# B&R Automation Studio project NAELD004C00R10L518F00 (part 22)

#### Visu_Layer.typ
```iecst
(*Common Layers*)

TYPE
	tyLyrC0001MotionStd : 	STRUCT
		tyBitmapOrigin : tyUIBitmap;
		tyBitmapPwr : tyUIBitmap;
		tyBitmapRst : tyUIBitmap;
		tyBitmapStop : tyUIBitmap;
		tyBitmapMc : tyUIBitmap;
		tyBtnPosLmtSen : tyUIBtn;
		tyBtnNegLmtSen : tyUIBtn;
		tyBtnJogPos : tyUIBtn;
		tyBtnJogNeg : tyUIBtn;
		tyBtnMovAbs : tyUIBtn;
		tyBtnMovRel : tyUIBtn;
		tyBtnOrigin : tyUIBtn;
		tyBtnPwr : tyUIBtn;
		tyBtnRst : tyUIBtn;
		tyBtnStop : tyUIBtn;
		tyNumCurrPos : tyUINum;
		tyNumErrCode : tyUINum;
		tyNumNomSpd : tyUINum;
		tyNumSlwSpd : tyUINum;
		tyNumStepSize : tyUINum;
		tyNumTargetPos : tyUINum;
		tyStringStat : tyUILString;
	END_STRUCT;
	tyLyrC0001MotionStdAW : 	STRUCT
		tyBitmapOrigin : tyUIBitmap;
		tyBitmapPwr : tyUIBitmap;
		tyBitmapRst : tyUIBitmap;
		tyBitmapStop : tyUIBitmap;
		tyBitmapMc : tyUIBitmap;
		tyBtnOpenLmtSen : tyUIBtn;
		tyBtnCloseLmtSen : tyUIBtn;
		tyBtnJogOpen : tyUIBtn;
		tyBtnJogClose : tyUIBtn;
		tyBtnMovAbs : tyUIBtn;
		tyBtnMovRel : tyUIBtn;
		tyBtnOrigin : tyUIBtn;
		tyBtnPwr : tyUIBtn;
		tyBtnRst : tyUIBtn;
		tyBtnStop : tyUIBtn;
		tyNumCurrPos : tyUINum;
		tyNumErrCode : tyUINum;
		tyNumNomSpd : tyUINum;
		tyNumSlwSpd : tyUINum;
		tyNumStepSize : tyUINum;
		tyNumTargetPos : tyUINum;
		tyStringStat : tyUILString;
	END_STRUCT;
	tyLyrC0001MotionStdLifter : 	STRUCT
		tyBitmapOrigin : tyUIBitmap;
		tyBitmapPwr : tyUIBitmap;
		tyBitmapRst : tyUIBitmap;
		tyBitmapStop : tyUIBitmap;
		tyBitmapMc : tyUIBitmap;
		tyBtnUpLmtSen : tyUIBtn;
		tyBtnDownLmtSen : tyUIBtn;
		tyBtnJogUp : tyUIBtn;
		tyBtnJogDown : tyUIBtn;
		tyBtnMovAbs : tyUIBtn;
		tyBtnMovRel : tyUIBtn;
		tyBtnOrigin : tyUIBtn;
		tyBtnPwr : tyUIBtn;
		tyBtnRst : tyUIBtn;
		tyBtnStop : tyUIBtn;
		tyNumCurrPos : tyUINum;
		tyNumErrCode : tyUINum;
		tyNumNomSpd : tyUINum;
		tyNumSlwSpd : tyUINum;
		tyNumStepSize : tyUINum;
		tyNumTargetPos : tyUINum;
		tyStringStat : tyUILString;
	END_STRUCT;
	tyLyrC0001MotionStdTrav : 	STRUCT
		tyBitmapOrigin : tyUIBitmap;
		tyBitmapPwr : tyUIBitmap;
		tyBitmapRst : tyUIBitmap;
		tyBitmapStop : tyUIBitmap;
		tyBitmapMc : tyUIBitmap;
		tyBtnFrontLmtSen : tyUIBtn;
		tyBtnRearLmtSen : tyUIBtn;
		tyBtnJogFront : tyUIBtn;
		tyBtnJogRear : tyUIBtn;
		tyBtnMovAbs : tyUIBtn;
		tyBtnMovRel : tyUIBtn;
		tyBtnOrigin : tyUIBtn;
		tyBtnPwr : tyUIBtn;
		tyBtnRst : tyUIBtn;
		tyBtnStop : tyUIBtn;
		tyNumCurrPos : tyUINum;
		tyNumErrCode : tyUINum;
		tyNumNomSpd : tyUINum;
		tyNumSlwSpd : tyUINum;
		tyNumStepSize : tyUINum;
		tyNumTargetPos : tyUINum;
		tyStringStat : tyUILString;
	END_STRUCT;
	tyLyrC0002FullMask : 	STRUCT
		tyLyr : tyUILyr;
		tyBtnMask : tyUIBtn;
	END_STRUCT;
	tyLyrC0003DualMask : 	STRUCT
		tyBtnLeftMask : tyUIBtn;
		tyBtnRgtMask : tyUIBtn;
		tyLyr : tyUILyr;
	END_STRUCT;
	tyLyrC0004Navi : 	STRUCT
		tyBtnLeft : tyUIBtn;
		tyBtnRgt : tyUIBtn;
		tyBtnBack : tyUIBtn;
		tyBitmapPageDisp : tyUIBitmap;
		tyLyr : tyUILyr;
	END_STRUCT;
	tyLyrC0005Main : 	STRUCT
		tyBtnNotification : tyUIBtn;
		tyBtnHome : tyUIBtn;
		tyBtnBuzzer : tyUIBtn;
		tyBtnStart : tyUIBtn;
		tyBtnStop : tyUIBtn;
		tyBtnStep : tyUIBtn;
		tyBtnReset : tyUIBtn;
		tyBitmapStatBar : tyUIBitmap;
		tyHotspotNaviStart : tyUIHotspot;
		tyBtnAlarm : tyUIBtn;
	END_STRUCT;
	tyLyrC0006Set : 	STRUCT
		tyBtnSave : tyUIBtn;
		tyLyr : tyUILyr;
	END_STRUCT;
	tyLyrC0007Notif : 	STRUCT
		tyTxtUsrLv : tyUITxt;
		tyTxtLFMc : tyUITxt;
		tyHotspotClose : tyUIHotspot;
		tyStringUsrNm : tyUIString;
		tyHotspotShowInfo : tyUIHotspot;
		tyBitmapShowInfo : tyUIBitmap;
		tyLyr : tyUILyr;
	END_STRUCT;
	tyLyrC0008MsgBox : 	STRUCT
		tyBitmapIcon : tyUIBitmap;
		tyBtnNo : tyUIBtn;
		tyBtnYes : tyUIBtn;
		tyLyr : tyUILyr;
		tyTxtWO_sLogMessage : tyUILString;
		tyTxtMsg : tyUITxt;
		tyTxtTitle : tyUITxt;
	END_STRUCT;
	tyLyrC0009Info : 	STRUCT
		tyStringInfo : tyUILString;
		tyHotspotClose : tyUIHotspot;
		tyLyr : tyUILyr;
	END_STRUCT;
	tyLyrC0010RcyMsg : 	STRUCT
		tyTxtMsg : tyUILString;
		tyHotspotClose : tyUIHotspot;
		tyLyr : tyUILyr;
	END_STRUCT;
	tyLyrC0011RcpPopUp : 	STRUCT
		tyStringInfo : tyUILString;
		tyHotspotClose : tyUIHotspot;
		tyLyr : tyUILyr;
	END_STRUCT;
END_TYPE

(**)
(**)
(*Pages*)

TYPE
	tyLyrP0000SSaver : 	STRUCT
		tyTxtMcStat : tyUITxt;
		tyTxtMcNm : tyUILString;
		tyBitmapStat : tyUIBitmap;
	END_STRUCT;
END_TYPE

(**)

TYPE
	tyLyrP0001Startup : 	STRUCT
		tyBarGraphStartup : tyUIBarGraph;
		tyTxtStartupStat : tyUITxt;
	END_STRUCT;
	tyLyrP0001Initial : 	STRUCT
		tyLyr : tyUILyr;
	END_STRUCT;
END_TYPE

(**)

TYPE
	tyLyrP0002Menu : 	STRUCT
		tyBtnAlm : tyUIBtn;
		tyBtnCommCtrl : tyUIBtn;
		tyBtnGenInput : tyUIBtn;
		tyBtnGenOutput : tyUIBtn;
		tyBtnLang : tyUIBtn;
		tyBtnLFCtrl : tyUIBtn;
		tyBtnLFSet : tyUIBtn;
		tyBtnLogin : tyUIBtn;
		tyBtnMcInfo : tyUIBtn;
		tyBtnMcSet : tyUIBtn;
		tyBtnMnlRst : tyUIBtn;
		tyBtnMovCtrl : tyUIBtn;
		tyBtnOpt : tyUIBtn;
		tyBtnProdSel : tyUIBtn;
		tyBtnProdSet : tyUIBtn;
		tyBtnMagInfo : tyUIBtn;
		tyBtnMagSet : tyUIBtn;
		tyBtnMagSel : tyUIBtn;
		tyBtnSimu : tyUIBtn;
		tyBtnUsrMgmt : tyUIBtn;
		tyBitmapMaskProdSetLCS : tyUIBitmap;
		tyHotspotProdSel : tyUIHotspot;
		tyHotspotMagSel : tyUIHotspot;
		tyBitmapGen : tyUIBitmap;
		tyBitmapSet : tyUIBitmap;
		tyBtnHotspotActSimu : tyUIBtn;
	END_STRUCT;
END_TYPE

(**)

TYPE
	tyLyrP0100Login : 	STRUCT
		tyStringUsrNm : tyUIString;
		tyStringPw : tyUIString;
		tyBtnLogin : tyUIBtn;
		tyHotspotBypassLogin : tyUIHotspot;
		tyLyr : tyUILyr;
	END_STRUCT;
	tyLyrP0100Logout : 	STRUCT
		tyBtnLogout : tyUIBtn;
		tyLyr : tyUILyr;
	END_STRUCT;
END_TYPE

(**)

TYPE
	tyLyrP0200OpsGen : 	STRUCT
		tyBtnAccDat : tyUIBtn;
		tyBitmapAccDat : tyUIBitmap;
		tyHotspotOpsTravLifter : tyUIHotspot;
		tyHotspotOps2Mag1 : tyUIHotspot;
		tyHotspotOps2Mag2 : tyUIHotspot;
		tyHotspotOpsTravLifterRToL : tyUIHotspot;
		tyHotspotOps2Mag1RToL : tyUIHotspot;
		tyHotspotOps2Mag2RToL : tyUIHotspot;
		tyHotspotOps3Mag1 : tyUIHotspot;
		tyHotspotOps3Mag2 : tyUIHotspot;
		tyHotspotOps3Mag3 : tyUIHotspot;
		tyHotspotOps4Mag1 : tyUIHotspot;
		tyHotspotOps4Mag2 : tyUIHotspot;
		tyHotspotOps4Mag3 : tyUIHotspot;
		tyHotspotOps4Mag4 : tyUIHotspot;
		tyHotspotOpsAIV : tyUIHotspot;
		tyHotspotOpsMagInfo : tyUIHotspot;
		tyNumMinSltRangeRear : tyUINum;
		tyNumMaxSltRangeRear : tyUINum;
		tyNumPitchRear : tyUINum;
		tyNumMinSltRange : tyUINum;
		tyNumMaxSltRange : tyUINum;
		tyNumPitch : tyUINum;
		tyTxtMagSlt : tyUITxt;
		tyNumMag1AvlQty : tyUINum;
		tyNumMag2AvlQty : tyUINum;
		tyNumMag3AvlQty : tyUINum;
		tyNumMag4AvlQty : tyUINum;
		tyNumMag1TtlSlt : tyUINum;
		tyNumMag2TtlSlt : tyUINum;
		tyNumMag3TtlSlt : tyUINum;
		tyNumMag4TtlSlt : tyUINum;
		tyHotspotAlm : tyUIHotspot;
		a_tyStringAlm : ARRAY[1..c_uiP0200TableSize]OF tyUILString;
		a_tyHotspotRcyMsg : ARRAY[1..c_uiP0200TableSize]OF tyUIHotspot;
		tyBitmapDSIn : tyUIBitmap;
		tyBitmapDSOut : tyUIBitmap;
		tyBitmapDSIn1 : tyUIBitmap;
		tyBitmapDSOut1 : tyUIBitmap;
		tyBitmapMc : tyUIBitmap;
		tyBitmapPCB : tyUIBitmap;
		tyBitmapDir1 : tyUIBitmap;
		tyBitmapDir2 : tyUIBitmap;
		tyTxtMag3Slt : tyUITxt;
		tyTxtBackslash3 : tyUITxt;
		tyTxtMag4Slt : tyUITxt;
		tyTxtBackslash4 : tyUITxt;
		tyTxtLane : tyUITxt;
		tyTxtLane1 : tyUITxt;
		tyBitmapDSAComm : tyUIBitmap;
		tyBitmapDSAComm1 : tyUIBitmap;
		tyHotspotDSAVSMEMA : tyUIHotspot;
		tyHotspotDSAVSMEMA1 : tyUIHotspot;
		tyTxtLdrInActiveCtrl : tyUITxt;
		tyBitmapWarningLF : tyUIBitmap;
		tyBitmapBarCodeScan : tyUIBitmap;
		tyBtnBarCodeScan : tyUIBtn;
		tyBtnTrolleyUnlck1 : tyUIBtn;
		tyBtnTrolleyUnlck2 : tyUIBtn;
	END_STRUCT;
	tyLyrP0200OpsDSCommB : 	STRUCT
		tyBitmapIn : tyUIBitmap;
		tyBitmapOut : tyUIBitmap;
		tyHotspotDSBVSMEMA : tyUIHotspot;
		tyBitmapDSBComm : tyUIBitmap;
		tyBitmapIn1 : tyUIBitmap;
		tyBitmapOut1 : tyUIBitmap;
		tyHotspotDSBVSMEMA1 : tyUIHotspot;
		tyBitmapDSBComm1 : tyUIBitmap;
		tyTxtLane : tyUITxt;
		tyTxtLane1 : tyUITxt;
		tyLyr : tyUILyr;
	END_STRUCT;
	tyLyrP0200OpsDSAVSMEMA : 	STRUCT
		tyBtnNom : tyUIBtn;
		tyBtnStat : tyUIBtn;
		tyLyr : tyUILyr;
	END_STRUCT;
	tyLyrP0200OpsDSBVSMEMA : 	STRUCT
		tyBtnNom : tyUIBtn;
		tyBtnStat : tyUIBtn;
		tyLyr : tyUILyr;
	END_STRUCT;
	tyLyrP0200OpsBypsInitConv : 	STRUCT
		tyBtnBypsInitConv : tyUIBtn;
		tyHotspotClose : tyUIHotspot;
		tyLyr : tyUILyr;
	END_STRUCT;
	tyLyrP0200OpsBarCodeScan : 	STRUCT  (*LMC scnner*)
		tyStringBarCode : tyUIString;
		tyStringWorkOrder : tyUIString;
		tyBtnUSBConnect : tyUIBtn;
		tyBtnOK : tyUIBtn;
		tyBtnCancel : tyUIBtn;
		tyLyr : tyUILyr;
	END_STRUCT;
END_TYPE

(**)

TYPE
	tyLyrP0201OpsTravLif : 	STRUCT
		tyBtnAccDat : tyUIBtn;
		tyBtnChgParam : tyUIBtn;
		tyHotspotIOMonitor : tyUIHotspot;
		tyBitmapAccDat : tyUIBitmap;
		tyTxtMod : tyUITxt;
		tyTxtWidth : tyUITxt;
		tyNumWidth : tyUINum;
		tyNumWidth2 : tyUINum;
		tyStringMcStat : tyUILString;
		tyStringProdNm : tyUILString;
		tyNumMinSltRange : tyUINum;
		tyNumMaxSltRange : tyUINum;
		tyNumPitch : tyUINum;
		tyNumMinSltRangeRear : tyUINum;
		tyNumMaxSltRangeRear : tyUINum;
		tyNumPitchRear : tyUINum;
		tyBtnToptoBtm : tyUIBtn;
		tyBitmapPCB : tyUIBitmap;
		tyBitmapMc : tyUIBitmap;
		tyTxtLdrInActiveCtrl : tyUITxt;
		tyBitmapWarningLF : tyUIBitmap;
		tyHotspotShowLRcp : tyUIHotspot;
		tyLyrProdRear : tyUILyr;
		tyNumMtrPshrExtSpd : tyUINum;
		tyNumMtrPshrExtTorq : tyUINum;
		tyNumPshrOffset : tyUINum;
	END_STRUCT;
	tyLyrP0201OpsTravLifIOMonitor : 	STRUCT
		tyHotspotClose : tyUIHotspot;
		tyBtnSafetyRlySig : tyUIBtn;
		tyBtnEStop : tyUIBtn;
		tyBtnCoverSWSig : tyUIBtn;
		tyBtnSafetyRlyRst : tyUIBtn;
		tyBtnTLGreen : tyUIBtn;
		tyBtnTLRed : tyUIBtn;
		tyBtnTLAmber : tyUIBtn;
		tyBtnBuzzer : tyUIBtn;
		tyBtnDSBA : tyUIBtn;
		tyBtnDSBB : tyUIBtn;
		tyBtnDBAA : tyUIBtn;
		tyBtnDBAB : tyUIBtn;
		tyBtnPullerExtRS : tyUIBtn;
		tyBtnPullerRetRS : tyUIBtn;
		tyBtnPullerRotCylHmRS : tyUIBtn;
		tyBtnPullerRotCylRmRS : tyUIBtn;
		tyBtnConvLftSen : tyUIBtn;
		tyBtnConvRgtSen : tyUIBtn;
		tyBtnConvClrSen : tyUIBtn;
		tyBtnLifterTmBeltSen : tyUIBtn;
		tyBtnLifterSafetyLmtSw1 : tyUIBtn;
		tyBtnLifterSafetyLmtSw2 : tyUIBtn;
		tyBtnMag1ClmpRS : tyUIBtn;
		tyBtnMag1UnclmpRS : tyUIBtn;
		tyBtnMag2ClmpRS : tyUIBtn;
		tyBtnMag2UnclmpRS : tyUIBtn;
		tyBtnMag3ClmpRS : tyUIBtn;
		tyBtnMag3UnclmpRS : tyUIBtn;
		tyBtnInletShutterOpenSen : tyUIBtn;
		tyBtnInletShutterCloseSen : tyUIBtn;
		tyBtnInletShutterOpenSen2 : tyUIBtn;
		tyBtnInletShutterCloseSen2 : tyUIBtn;
		tyBtnInletShutterOpenSen3 : tyUIBtn;
		tyBtnInletShutterCloseSen3 : tyUIBtn;
		tyBtnOutletShutterOpenSen : tyUIBtn;
		tyBtnOutletShutterCloseSen : tyUIBtn;
		tyBtnOutletShutterOpenSen2 : tyUIBtn;
		tyBtnOutletShutterCloseSen2 : tyUIBtn;
		tyBtnMag1PresentSen : tyUIBtn;
		tyBtnMag2PresentSen : tyUIBtn;
		tyBtnMag3PresentSen : tyUIBtn;
		tyBtnMag1ConvEntrySen : tyUIBtn;
		tyBtnMag2ConvEntrySen : tyUIBtn;
		tyBtnMag3ConvEntrySen : tyUIBtn;
		tyBtnMag1AIVInPosSen1 : tyUIBtn;
		tyBtnMag1AIVInPosSen2 : tyUIBtn;
		tyBtnMag2AIVInPosSen1 : tyUIBtn;
		tyBtnMag2AIVInPosSen2 : tyUIBtn;
		tyBtnMag3AIVInPosSen1 : tyUIBtn;
		tyBtnMag3AIVInPosSen2 : tyUIBtn;
		tyBtnMag1OrientationChkSen1 : tyUIBtn;
		tyBtnMag2OrientationChkSen1 : tyUIBtn;
		tyBtnMag3OrientationChkSen1 : tyUIBtn;
		tyBtnMag1OrientationChkSen2 : tyUIBtn;
		tyBtnMag2OrientationChkSen2 : tyUIBtn;
		tyBtnMag3OrientationChkSen2 : tyUIBtn;
		tyBtnPullerExtCtrl : tyUIBtn;
		tyBtnPullerRetCtrl : tyUIBtn;
		tyBtnRotPullerCtrl : tyUIBtn;
		tyBtnInShutterOpenCtrl : tyUIBtn;
		tyBtnInShutterCloseCtrl : tyUIBtn;
		tyBtnInShutterOpenCtrl2 : tyUIBtn;
		tyBtnInShutterCloseCtrl2 : tyUIBtn;
		tyBtnInShutterOpenCtrl3 : tyUIBtn;
		tyBtnInShutterCloseCtrl3 : tyUIBtn;
		tyBtnOutShutterOpenCtrl : tyUIBtn;
		tyBtnOutShutterCloseCtrl : tyUIBtn;
		tyBtnOutShutterOpenCtrl2 : tyUIBtn;
		tyBtnOutShutterCloseCtrl2 : tyUIBtn;
		tyBtnPullerConvMtrOn : tyUIBtn;
		tyBtnAntiJamSen : tyUIBtn;
		tyBtnRstCurtainSensor : tyUIBtn;
		tyBtnBypCurtainSensorCtrl : tyUIBtn;
		tyBtnBypCurtainSensorPB : tyUIBtn;
		tyBtnMagWidthChk : tyUIBtn;
		tyBtnUnlockSigDS : tyUIBtn;
		tyBtnSafetySigDS : tyUIBtn;
		tyBtnSftySglToUSDS : tyUIBtn;
		tyLyr : tyUILyr;
	END_STRUCT;
	tyLyrP0201OpsTravLifBypsInitConv : 	STRUCT
		tyBtnBypsInitConv : tyUIBtn;
		tyHotspotClose : tyUIHotspot;
		tyLyr : tyUILyr;
	END_STRUCT;
	tyLyrP0201OpsParam : 	STRUCT
		tyDrpDnMcMode : tyUIDrpDn;
		tyNumMinSlt : tyUINum;
		tyNumMaxSlt : tyUINum;
		tyNumPitch : tyUINum;
		tyBtnToptoBtm : tyUIBtn;
		tyNumMinSltRear : tyUINum;
		tyNumMaxSltRear : tyUINum;
		tyNumPitchRear : tyUINum;
		tyBtnToptoBtmRear : tyUIBtn;
		tyBtnSave : tyUIBtn;
		tyBtnCancel : tyUIBtn;
		tyNumMtrPshrExtSpd : tyUINum;
		tyNumMtrPshrExtTorq : tyUINum;
		tyNumPshrOffset : tyUINum;
		tyLyr : tyUILyr;
	END_STRUCT;
	tyLyrP0201OpsQueryBoardInfo : 	STRUCT
		tyBtnOk : tyUIBtn;
		tyBtnQueryBoardInfo : tyUIBtn;
		tyBtnCancel : tyUIBtn;
		tyBtnBarcodeScanner : tyUIBtn;
		tyStringTopBarcode : tyUILString;
		tyStringBottomBarcode : tyUILString;
		tyLyr : tyUILyr;
	END_STRUCT;
	tyLyrP0201OpsCurrWorkOrder : 	STRUCT
		tyBtnQuery : tyUIBtn;
		tyBtnExit : tyUIBtn;
		tyBtnDelete : tyUIBtn;
		tyStringWorkOrder : tyUILString;
		tyBtnQueryWorkOrderInfo : tyUIBtn;
		tyLyr : tyUILyr;
		tyBitmapMask : tyUIBitmap;
	END_STRUCT;
	tyLyrP0201OpsQueryWorkOrder : 	STRUCT
		tyBtnOk : tyUIBtn;
		tyBtnCancel : tyUIBtn;
		tyBtnBarcodeScanner : tyUIBtn;
		tyStringMagazineId : tyUILString;
		tyNumSlotId : tyUINum;
		tyStringBarcode : tyUILString;
		tyLyr : tyUILyr;
		tyBitmapMask : tyUIBitmap;
	END_STRUCT;
	tyLyrP0201OpsBarcodeScanner : 	STRUCT
		tyBtnOk : tyUIBtn;
		tyBtnCancel : tyUIBtn;
		tyStringBarcode : tyUILString;
		tyStringTopBarcode : tyUILString;
		tyStringTopBarcodeBK : tyUILString;
		tyStringBottomBarcode : tyUILString;
		tyStringBottomBarcodeBK : tyUILString;
		tyStringMagazineBarcode : tyUILString;
		tyStringMagazineBarcodeBK : tyUILString;
		tyStringPCBBarcode : tyUILString;
		tyStringPCBBarcodeBK : tyUILString;
		tyBtnTop : tyUIBtn;
		tyBtnBottom : tyUIBtn;
		tyBtnMagazine : tyUIBtn;
		tyBtnPCB : tyUIBtn;
		tyLyr : tyUILyr;
	END_STRUCT;
END_TYPE

(**)

TYPE
	tyLyrP0202Ops : 	STRUCT
		tyBtnAccDat : tyUIBtn;
		tyBtnChgParam : tyUIBtn;
		tyBitmapAccDat : tyUIBitmap;
		tyTxtMod : tyUITxt;
		tyTxtWidth : tyUITxt;
		tyNumWidth : tyUINum;
		tyNumWidth2 : tyUINum;
		tyTxtMag1Stat : tyUITxt;
		tyStringMcStat : tyUILString;
		tyHotspotIOMonitor : tyUIHotspot;
		tyHotspotMagInfo : tyUIHotspot;
		tyStringProdNm : tyUILString;
		tyNumMinSltRange : tyUINum;
		tyNumMaxSltRange : tyUINum;
		tyNumPitch : tyUINum;
		tyBtnToptoBtm : tyUIBtn;
		tyStringMagNm : tyUIString;
		tyTxtMagSlt : tyUITxt;
		tyNumMag1AvlQty : tyUINum;
		tyNumMag1TtlSlt : tyUINum;
		tyBitmapMc : tyUIBitmap;
		tyTxtLblAIV : tyUITxt;
		tyBtnAIVWifi : tyUIBtn;
		tyBtnChgMag : tyUIBtn;
		tyBitmapChgMag : tyUIBitmap;
		tyTxtLdrInActiveCtrl : tyUITxt;
		tyBitmapWarningLF : tyUIBitmap;
		tyHotspotShowLRcp : tyUIHotspot;
		tyBitmapUnloadMag : tyUIBitmap;
		tyBtnUnloadMag : tyUIBtn;
	END_STRUCT;
	tyLyrP0202IOMonitor : 	STRUCT
		tyHotspotClose : tyUIHotspot;
		tyBtnSafetyRlySig : tyUIBtn;
		tyBtnEStop : tyUIBtn;
		tyBtnCoverSWSig : tyUIBtn;
		tyBtnSafetyRlyRst : tyUIBtn;
		tyBtnTLGreen : tyUIBtn;
		tyBtnTLRed : tyUIBtn;
		tyBtnTLAmber : tyUIBtn;
		tyBtnBuzzer : tyUIBtn;
		tyBtnDSBA : tyUIBtn;
		tyBtnDSBB : tyUIBtn;
		tyBtnDBAA : tyUIBtn;
		tyBtnDBAB : tyUIBtn;
		tyBtnPullerExtRS : tyUIBtn;
		tyBtnPullerRetRS : tyUIBtn;
		tyBtnPullerRotCylHmRS : tyUIBtn;
		tyBtnPullerRotCylRmRS : tyUIBtn;
		tyBtnPullerOutSen : tyUIBtn;
		tyBtnPullerClrSen : tyUIBtn;
		tyBtnLifterTmBeltSen : tyUIBtn;
		tyBtnLimitSafetySw1 : tyUIBtn;
		tyBtnLimitSafetySw2 : tyUIBtn;
		tyBtnMag1FixedClmpRS : tyUIBtn;
		tyBtnMag1FixedUnclmpRS : tyUIBtn;
		tyBtnMag1RmtClmpRS : tyUIBtn;
		tyBtnMag1RmtUnclmpRS : tyUIBtn;
		tyBtnMag2FixedClmpRS : tyUIBtn;
		tyBtnMag2FixedUnclmpRS : tyUIBtn;
		tyBtnMag2RmtClmpRS : tyUIBtn;
		tyBtnMag2RmtUnclmpRS : tyUIBtn;
		tyBtnMag3FixedClmpRS : tyUIBtn;
		tyBtnMag3FixedUnclmpRS : tyUIBtn;
		tyBtnMag3RmtClmpRS : tyUIBtn;
		tyBtnMag3RmtUnclmpRS : tyUIBtn;
		tyBtnInletShutterOpenSen : tyUIBtn;
		tyBtnInletShutterCloseSen : tyUIBtn;
		tyBtnOutletShutterOpenSen : tyUIBtn;
		tyBtnOutletShutterCloseSen : tyUIBtn;
		tyBtnMag1PresentSen : tyUIBtn;
		tyBtnMag2PresentSen : tyUIBtn;
		tyBtnMag3PresentSen : tyUIBtn;
		tyBtnMag1ConvEntrySen : tyUIBtn;
		tyBtnMag2ConvEntrySen : tyUIBtn;
		tyBtnMag3ConvEntrySen : tyUIBtn;
		tyBtnMag1AIVInPosSen1 : tyUIBtn;
		tyBtnMag1AIVInPosSen2 : tyUIBtn;
		tyBtnMag2AIVInPosSen1 : tyUIBtn;
		tyBtnMag2AIVInPosSen2 : tyUIBtn;
		tyBtnMag3AIVInPosSen1 : tyUIBtn;
		tyBtnMag3AIVInPosSen2 : tyUIBtn;
		tyBtnMag1OrientationChkSen1 : tyUIBtn;
		tyBtnMag2OrientationChkSen1 : tyUIBtn;
		tyBtnMag3OrientationChkSen1 : tyUIBtn;
		tyBtnMag1OrientationChkSen2 : tyUIBtn;
		tyBtnMag2OrientationChkSen2 : tyUIBtn;
		tyBtnMag3OrientationChkSen2 : tyUIBtn;
		tyLyr : tyUILyr;
		tyBtnMag1FixedClampCtrl : tyUIBtn;
		tyBtnMag1RemoteClampCtrl : tyUIBtn;
		tyBtnMag1ConvMtrIn : tyUIBtn;
		tyBtnMag1ConvMtrOut : tyUIBtn;
		tyBtnSelUnclampRS : tyUIBtn;
		tyBtnHeightSen : tyUIBtn;
		tyBtnCAB717Sen : tyUIBtn;
		tyBtnMagSmallSen : tyUIBtn;
		tyBtnMagLargeSen : tyUIBtn;
		tyBtnMagSelClampCtrl : tyUIBtn;
		tyBtnMagDetSen : tyUIBtn;
		tyBtnSltLckSen : tyUIBtn;
		tyBtnTrllyExtRS : tyUIBtn;
		tyBtnTrllyPresentSen : tyUIBtn;
		tyBtnTrllyExtCtrl : tyUIBtn;
	END_STRUCT;
	tyLyrP0202BypsInitConv : 	STRUCT
		tyBtnBypsInitConv : tyUIBtn;
		tyHotspotClose : tyUIHotspot;
		tyLyr : tyUILyr;
	END_STRUCT;
	tyLyrP0202OpsParam : 	STRUCT
		tyDrpDnMcMode : tyUIDrpDn;
		tyNumMinSlt : tyUINum;
		tyNumMaxSlt : tyUINum;
		tyNumPitch : tyUINum;
		tyBtnToptoBtm : tyUIBtn;
		tyNumMinSltRear : tyUINum;
		tyNumMaxSltRear : tyUINum;
		tyNumPitchRear : tyUINum;
		tyBtnToptoBtmRear : tyUIBtn;
		tyBtnSave : tyUIBtn;
		tyBtnCancel : tyUIBtn;
		tyNumMtrPshrExtSpd : tyUINum;
		tyNumMtrPshrExtTorq : tyUINum;
		tyNumPshrOffset : tyUINum;
		tyLyr : tyUILyr;
	END_STRUCT;
END_TYPE

(**)

TYPE
	tyLyrP0203Ops : 	STRUCT
		tyBtnAccDat : tyUIBtn;
		tyBtnChgParam : tyUIBtn;
		tyHotspotIOMonitor : tyUIHotspot;
		tyBitmapAccDat : tyUIBitmap;
		tyTxtMod : tyUITxt;
		tyTxtWidth : tyUITxt;
		tyNumWidth2 : tyUINum;
		tyNumWidth : tyUINum;
		tyTxtMag2Stat : tyUITxt;
		tyStringMcStat : tyUILString;
		tyHotspotMagInfo : tyUIHotspot;
		tyStringProdNm : tyUILString;
		tyNumMinSltRange : tyUINum;
		tyNumMaxSltRange : tyUINum;
		tyNumPitch : tyUINum;
		tyBtnToptoBtm : tyUIBtn;
		tyStringMagNm : tyUIString;
		tyTxtMagSlt : tyUITxt;
		tyNumMag2AvlQty : tyUINum;
		tyNumMag2TtlSlt : tyUINum;
		tyBitmapMc : tyUIBitmap;
		tyTxtLblAIV : tyUITxt;
		tyBtnAIVWifi : tyUIBtn;
		tyBtnChgMag : tyUIBtn;
		tyBitmapChgMag : tyUIBitmap;
		tyTxtLdrInActiveCtrl : tyUITxt;
		tyBitmapWarningLF : tyUIBitmap;
		tyHotspotShowLRcp : tyUIHotspot;
		tyBitmapUnloadMag : tyUIBitmap;
		tyBtnUnloadMag : tyUIBtn;
	END_STRUCT;
	tyLyrP0203IOMonitor : 	STRUCT
		tyHotspotClose : tyUIHotspot;
		tyBtnSafetyRlySig : tyUIBtn;
		tyBtnEStop : tyUIBtn;
		tyBtnCoverSWSig : tyUIBtn;
		tyBtnSafetyRlyRst : tyUIBtn;
		tyBtnTLGreen : tyUIBtn;
		tyBtnTLRed : tyUIBtn;
		tyBtnTLAmber : tyUIBtn;
		tyBtnBuzzer : tyUIBtn;
		tyBtnDSBA : tyUIBtn;
		tyBtnDSBB : tyUIBtn;
		tyBtnDBAA : tyUIBtn;
		tyBtnDBAB : tyUIBtn;
		tyBtnPullerExtRS : tyUIBtn;
		tyBtnPullerRetRS : tyUIBtn;
		tyBtnPullerRotCylHmRS : tyUIBtn;
		tyBtnPullerRotCylRmRS : tyUIBtn;
		tyBtnPullerOutSen : tyUIBtn;
		tyBtnPullerClrSen : tyUIBtn;
		tyBtnLifterTmBeltSen : tyUIBtn;
		tyBtnLimitSafetySw1 : tyUIBtn;
		tyBtnLimitSafetySw2 : tyUIBtn;
		tyBtnMag1FixedClmpRS : tyUIBtn;
		tyBtnMag1FixedUnclmpRS : tyUIBtn;
		tyBtnMag1RmtClmpRS : tyUIBtn;
		tyBtnMag1RmtUnclmpRS : tyUIBtn;
		tyBtnMag2FixedClmpRS : tyUIBtn;
		tyBtnMag2FixedUnclmpRS : tyUIBtn;
		tyBtnMag2RmtClmpRS : tyUIBtn;
		tyBtnMag2RmtUnclmpRS : tyUIBtn;
		tyBtnMag3FixedClmpRS : tyUIBtn;
		tyBtnMag3FixedUnclmpRS : tyUIBtn;
		tyBtnMag3RmtClmpRS : tyUIBtn;
		tyBtnMag3RmtUnclmpRS : tyUIBtn;
		tyBtnInletShutterOpenSen : tyUIBtn;
		tyBtnInletShutterCloseSen : tyUIBtn;
		tyBtnOutletShutterOpenSen : tyUIBtn;
		tyBtnOutletShutterCloseSen : tyUIBtn;
		tyBtnMag1PresentSen : tyUIBtn;
		tyBtnMag2PresentSen : tyUIBtn;
		tyBtnMag3PresentSen : tyUIBtn;
		tyBtnMag1ConvEntrySen : tyUIBtn;
		tyBtnMag2ConvEntrySen : tyUIBtn;
		tyBtnMag3ConvEntrySen : tyUIBtn;
		tyBtnMag1AIVInPosSen1 : tyUIBtn;
		tyBtnMag1AIVInPosSen2 : tyUIBtn;
		tyBtnMag2AIVInPosSen1 : tyUIBtn;
		tyBtnMag2AIVInPosSen2 : tyUIBtn;
		tyBtnMag3AIVInPosSen1 : tyUIBtn;
		tyBtnMag3AIVInPosSen2 : tyUIBtn;
		tyBtnMag1OrientationChkSen1 : tyUIBtn;
		tyBtnMag2OrientationChkSen1 : tyUIBtn;
		tyBtnMag3OrientationChkSen1 : tyUIBtn;
		tyBtnMag1OrientationChkSen2 : tyUIBtn;
		tyBtnMag2OrientationChkSen2 : tyUIBtn;
		tyBtnMag3OrientationChkSen2 : tyUIBtn;
		tyLyr : tyUILyr;
		tyBtnMag2FixedClampCtrl : tyUIBtn;
		tyBtnMag2RemoteClampCtrl : tyUIBtn;
		tyBtnMag2ConvMtrIn : tyUIBtn;
		tyBtnMag2ConvMtrOut : tyUIBtn;
		tyBtnSelUnclampRS : tyUIBtn;
		tyBtnHeightSen : tyUIBtn;
		tyBtnCAB717Sen : tyUIBtn;
		tyBtnMagSmallSen : tyUIBtn;
		tyBtnMagLargeSen : tyUIBtn;
		tyBtnMagSelClampCtrl : tyUIBtn;
		tyBtnMagDetSen : tyUIBtn;
		tyBtnSltLckSen : tyUIBtn;
		tyBtnTrllyExtRS : tyUIBtn;
		tyBtnTrllyPresentSen : tyUIBtn;
		tyBtnTrllyExtCtrl : tyUIBtn;
	END_STRUCT;
	tyLyrP0203BypsInitConv : 	STRUCT
		tyBtnBypsInitConv : tyUIBtn;
		tyHotspotClose : tyUIHotspot;
		tyLyr : tyUILyr;
	END_STRUCT;
	tyLyrP0203OpsParam : 	STRUCT
		tyDrpDnMcMode : tyUIDrpDn;
		tyNumMinSlt : tyUINum;
		tyNumMaxSlt : tyUINum;
		tyNumPitch : tyUINum;
		tyBtnToptoBtm : tyUIBtn;
		tyNumMinSltRear : tyUINum;
		tyNumMaxSltRear : tyUINum;
		tyNumPitchRear : tyUINum;
		tyBtnToptoBtmRear : tyUIBtn;
		tyBtnSave : tyUIBtn;
		tyBtnCancel : tyUIBtn;
		tyNumMtrPshrExtSpd : tyUINum;
		tyNumMtrPshrExtTorq : tyUINum;
		tyNumPshrOffset : tyUINum;
		tyLyr : tyUILyr;
	END_STRUCT;
END_TYPE

(**)

TYPE
	tyLyrP0204Ops : 	STRUCT
		tyBtnAccDat : tyUIBtn;
		tyBtnChgParam : tyUIBtn;
		tyHotspotIOMonitor : tyUIHotspot;
		tyBitmapAccDat : tyUIBitmap;
		tyTxtMod : tyUITxt;
		tyTxtWidth : tyUITxt;
		tyNumWidth : tyUINum;
		tyNumWidth2 : tyUINum;
		tyTxtMag3Stat : tyUITxt;
		tyStringMcStat : tyUILString;
		tyHotspotMagInfo : tyUIHotspot;
		tyStringProdNm : tyUILString;
		tyNumMinSltRange : tyUINum;
		tyNumMaxSltRange : tyUINum;
		tyNumPitch : tyUINum;
		tyBtnToptoBtm : tyUIBtn;
		tyStringMagNm : tyUIString;
		tyTxtMagSlt : tyUITxt;
		tyNumMag3AvlQty : tyUINum;
		tyNumMag3TtlSlt : tyUINum;
		tyBitmapMc : tyUIBitmap;
		tyTxtLblAIV : tyUITxt;
		tyBtnAIVWifi : tyUIBtn;
		tyBtnChgMag : tyUIBtn;
		tyBitmapChgMag : tyUIBitmap;
		tyTxtLdrInActiveCtrl : tyUITxt;
		tyBitmapWarningLF : tyUIBitmap;
		tyHotspotShowLRcp : tyUIHotspot;
		tyBitmapUnloadMag : tyUIBitmap;
		tyBtnUnloadMag : tyUIBtn;
	END_STRUCT;
	tyLyrP0204IOMonitor : 	STRUCT
		tyHotspotClose : tyUIHotspot;
		tyBtnSafetyRlySig : tyUIBtn;
		tyBtnEStop : tyUIBtn;
		tyBtnCoverSWSig : tyUIBtn;
		tyBtnSafetyRlyRst : tyUIBtn;
		tyBtnTLGreen : tyUIBtn;
		tyBtnTLRed : tyUIBtn;
		tyBtnTLAmber : tyUIBtn;
		tyBtnBuzzer : tyUIBtn;
		tyBtnDSBA : tyUIBtn;
		tyBtnDSBB : tyUIBtn;
		tyBtnDBAA : tyUIBtn;
		tyBtnDBAB : tyUIBtn;
		tyBtnPullerExtRS : tyUIBtn;
		tyBtnPullerRetRS : tyUIBtn;
		tyBtnPullerRotCylHmRS : tyUIBtn;
		tyBtnPullerRotCylRmRS : tyUIBtn;
		tyBtnPullerOutSen : tyUIBtn;
		tyBtnPullerClrSen : tyUIBtn;
		tyBtnLifterTmBeltSen : tyUIBtn;
		tyBtnLimitSafetySw1 : tyUIBtn;
		tyBtnLimitSafetySw2 : tyUIBtn;
		tyBtnMag1FixedClmpRS : tyUIBtn;
		tyBtnMag1FixedUnclmpRS : tyUIBtn;
		tyBtnMag1RmtClmpRS : tyUIBtn;
		tyBtnMag1RmtUnclmpRS : tyUIBtn;
		tyBtnMag2FixedClmpRS : tyUIBtn;
		tyBtnMag2FixedUnclmpRS : tyUIBtn;
		tyBtnMag2RmtClmpRS : tyUIBtn;
		tyBtnMag2RmtUnclmpRS : tyUIBtn;
		tyBtnMag3FixedClmpRS : tyUIBtn;
		tyBtnMag3FixedUnclmpRS : tyUIBtn;
		tyBtnMag3RmtClmpRS : tyUIBtn;
		tyBtnMag3RmtUnclmpRS : tyUIBtn;
		tyBtnInletShutterOpenSen : tyUIBtn;
		tyBtnInletShutterCloseSen : tyUIBtn;
		tyBtnOutletShutterOpenSen : tyUIBtn;
		tyBtnOutletShutterCloseSen : tyUIBtn;
		tyBtnMag1PresentSen : tyUIBtn;
		tyBtnMag2PresentSen : tyUIBtn;
		tyBtnMag3PresentSen : tyUIBtn;
		tyBtnMag1ConvEntrySen : tyUIBtn;
		tyBtnMag2ConvEntrySen : tyUIBtn;
		tyBtnMag3ConvEntrySen : tyUIBtn;
		tyBtnMag1AIVInPosSen1 : tyUIBtn;
		tyBtnMag1AIVInPosSen2 : tyUIBtn;
		tyBtnMag2AIVInPosSen1 : tyUIBtn;
		tyBtnMag2AIVInPosSen2 : tyUIBtn;
		tyBtnMag3AIVInPosSen1 : tyUIBtn;
		tyBtnMag3AIVInPosSen2 : tyUIBtn;
		tyBtnMag1OrientationChkSen1 : tyUIBtn;
		tyBtnMag2OrientationChkSen1 : tyUIBtn;
		tyBtnMag3OrientationChkSen1 : tyUIBtn;
		tyBtnMag1OrientationChkSen2 : tyUIBtn;
		tyBtnMag2OrientationChkSen2 : tyUIBtn;
		tyBtnMag3OrientationChkSen2 : tyUIBtn;
		tyLyr : tyUILyr;
		tyBtnMag3FixedClampCtrl : tyUIBtn;
		tyBtnMag3RemoteClampCtrl : tyUIBtn;
		tyBtnMag3ConvMtrIn : tyUIBtn;
		tyBtnMag3ConvMtrOut : tyUIBtn;
		tyBtnSelUnclampRS : tyUIBtn;
		tyBtnHeightSen : tyUIBtn;
		tyBtnCAB717Sen : tyUIBtn;
		tyBtnMagSmallSen : tyUIBtn;
		tyBtnMagLargeSen : tyUIBtn;
		tyBtnMagSelClampCtrl : tyUIBtn;
		tyBtnMagDetSen : tyUIBtn;
	END_STRUCT;
	tyLyrP0204BypsInitConv : 	STRUCT
		tyBtnBypsInitConv : tyUIBtn;
		tyHotspotClose : tyUIHotspot;
		tyLyr : tyUILyr;
	END_STRUCT;
	tyLyrP0204OpsParam : 	STRUCT
		tyDrpDnMcMode : tyUIDrpDn;
		tyNumMinSlt : tyUINum;
		tyNumMaxSlt : tyUINum;
		tyNumPitch : tyUINum;
		tyBtnToptoBtm : tyUIBtn;
		tyNumMinSltRear : tyUINum;
		tyNumMaxSltRear : tyUINum;
		tyNumPitchRear : tyUINum;
		tyBtnToptoBtmRear : tyUIBtn;
		tyBtnSave : tyUIBtn;
		tyBtnCancel : tyUIBtn;
		tyNumMtrPshrExtSpd : tyUINum;
		tyNumMtrPshrExtTorq : tyUINum;
		tyNumPshrOffset : tyUINum;
		tyLyr : tyUILyr;
	END_STRUCT;
END_TYPE

(**)

TYPE
	tyLyrP0205IOMonitor : 	STRUCT
		tyHotspotClose : tyUIHotspot;
		tyBitmapMc : tyUIBitmap;
		tyBitmapAIVErr1 : tyUIBitmap;
		tyBitmapAIVErr2 : tyUIBitmap;
		tyBitmapAIVErr3 : tyUIBitmap;
		tyBitmapAIVErr4 : tyUIBitmap;
		tyBitmapAIVRdy1 : tyUIBitmap;
		tyBitmapAIVRdy2 : tyUIBitmap;
		tyBitmapAIVRdy3 : tyUIBitmap;
		tyBitmapAIVRdy4 : tyUIBitmap;
		tyBitmapAIVAvail1 : tyUIBitmap;
		tyBitmapAIVAvail2 : tyUIBitmap;
		tyBitmapAIVAvail3 : tyUIBitmap;
		tyBitmapAIVAvail4 : tyUIBitmap;
		tyBitmapAIVSLarge1 : tyUIBitmap;
		tyBitmapAIVSLarge2 : tyUIBitmap;
		tyBitmapAIVSLarge3 : tyUIBitmap;
		tyBitmapAIVSLarge4 : tyUIBitmap;
		tyBtnAIVSotRCVOk1 : tyUIBtn;
		tyBtnAIVSotRCVOk2 : tyUIBtn;
		tyBtnAIVSotRCVOk3 : tyUIBtn;
		tyBtnAIVSotRCVOk4 : tyUIBtn;
		tyBtnReqAIVToBring1 : tyUIBtn;
		tyBtnReqAIVToBring2 : tyUIBtn;
		tyBtnReqAIVToBring3 : tyUIBtn;
		tyBtnReqAIVToBring4 : tyUIBtn;
		tyBtnReqAIVToGet1 : tyUIBtn;
		tyBtnReqAIVToGet2 : tyUIBtn;
		tyBtnReqAIVToGet3 : tyUIBtn;
		tyBtnReqAIVToGet4 : tyUIBtn;
		tyBitmapMagErr1 : tyUIBitmap;
		tyBitmapMagErr2 : tyUIBitmap;
		tyBitmapMagErr3 : tyUIBitmap;
		tyBitmapMagErr4 : tyUIBitmap;
		tyBitmapMagRdy1 : tyUIBitmap;
		tyBitmapMagRdy2 : tyUIBitmap;
		tyBitmapMagRdy3 : tyUIBitmap;
		tyBitmapMagRdy4 : tyUIBitmap;
		tyBitmapMagAvail1 : tyUIBitmap;
		tyBitmapMagAvail2 : tyUIBitmap;
		tyBitmapMagAvail3 : tyUIBitmap;
		tyBitmapMagAvail4 : tyUIBitmap;
		tyBitmapMagSLarge1 : tyUIBitmap;
		tyBitmapMagSLarge2 : tyUIBitmap;
		tyBitmapMagSLarge3 : tyUIBitmap;
		tyBitmapMagSLarge4 : tyUIBitmap;
		tyBtnMESActive : tyUIBtn;
		tyStringMesName : tyUILString;
		tyLyr12 : tyUILyr;
		tyLyr3 : tyUILyr;
		tyLyr4 : tyUILyr;
		tyTxtAIVCommProtocol : tyUITxt;
	END_STRUCT;
END_TYPE

(**)

TYPE
	tyLyrP0206Ops : 	STRUCT
		tyBtnAccDat : tyUIBtn;
		tyBtnChgParam : tyUIBtn;
		tyHotspotIOMonitor : tyUIHotspot;
		tyBitmapAccDat : tyUIBitmap;
		tyTxtMod : tyUITxt;
		tyTxtWidth : tyUITxt;
		tyNumWidth : tyUINum;
		tyNumWidth2 : tyUINum;
		tyTxtMag4Stat : tyUITxt;
		tyStringMcStat : tyUILString;
		tyHotspotMagInfo : tyUIHotspot;
		tyStringProdNm : tyUILString;
		tyNumMinSltRange : tyUINum;
		tyNumMaxSltRange : tyUINum;
		tyNumPitch : tyUINum;
		tyBtnToptoBtm : tyUIBtn;
		tyStringMagNm : tyUIString;
		tyTxtMagSlt : tyUITxt;
		tyNumMag4AvlQty : tyUINum;
		tyNumMag4TtlSlt : tyUINum;
		tyBitmapMc : tyUIBitmap;
		tyTxtLblAIV : tyUITxt;
		tyBtnAIVWifi : tyUIBtn;
		tyBtnChgMag : tyUIBtn;
		tyBitmapChgMag : tyUIBitmap;
		tyTxtLdrInActiveCtrl : tyUITxt;
		tyBitmapWarningLF : tyUIBitmap;
		tyHotspotShowLRcp : tyUIHotspot;
		tyBitmapUnloadMag : tyUIBitmap;
		tyBtnUnloadMag : tyUIBtn;
	END_STRUCT;
	tyLyrP0206IOMonitor : 	STRUCT
		tyHotspotClose : tyUIHotspot;
		tyBtnSafetyRlySig : tyUIBtn;
		tyBtnEStop : tyUIBtn;
		tyBtnCoverSWSig : tyUIBtn;
		tyBtnSafetyRlyRst : tyUIBtn;
		tyBtnTLGreen : tyUIBtn;
		tyBtnTLRed : tyUIBtn;
		tyBtnTLAmber : tyUIBtn;
		tyBtnBuzzer : tyUIBtn;
		tyBtnDSBA : tyUIBtn;
		tyBtnDSBB : tyUIBtn;
		tyBtnDBAA : tyUIBtn;
		tyBtnDBAB : tyUIBtn;
		tyBtnPullerExtRS : tyUIBtn;
		tyBtnPullerRetRS : tyUIBtn;
		tyBtnPullerRotCylHmRS : tyUIBtn;
		tyBtnPullerRotCylRmRS : tyUIBtn;
		tyBtnPullerOutSen : tyUIBtn;
		tyBtnPullerClrSen : tyUIBtn;
		tyBtnLifterTmBeltSen : tyUIBtn;
		tyBtnLimitSafetySw1 : tyUIBtn;
		tyBtnLimitSafetySw2 : tyUIBtn;
		tyBtnMag1FixedClmpRS : tyUIBtn;
		tyBtnMag1FixedUnclmpRS : tyUIBtn;
		tyBtnMag1RmtClmpRS : tyUIBtn;
		tyBtnMag1RmtUnclmpRS : tyUIBtn;
		tyBtnMag2FixedClmpRS : tyUIBtn;
		tyBtnMag2FixedUnclmpRS : tyUIBtn;
		tyBtnMag2RmtClmpRS : tyUIBtn;
		tyBtnMag2RmtUnclmpRS : tyUIBtn;
		tyBtnMag3FixedClmpRS : tyUIBtn;
		tyBtnMag3FixedUnclmpRS : tyUIBtn;
		tyBtnMag3RmtClmpRS : tyUIBtn;
		tyBtnMag3RmtUnclmpRS : tyUIBtn;
		tyBtnMag4FixedClmpRS : tyUIBtn;
		tyBtnMag4FixedUnclmpRS : tyUIBtn;
		tyBtnMag4RmtClmpRS : tyUIBtn;
		tyBtnMag4RmtUnclmpRS : tyUIBtn;
		tyBtnInletShutterOpenSen : tyUIBtn;
		tyBtnInletShutterCloseSen : tyUIBtn;
		tyBtnOutletShutterOpenSen : tyUIBtn;
		tyBtnOutletShutterCloseSen : tyUIBtn;
		tyBtnMag1PresentSen : tyUIBtn;
		tyBtnMag2PresentSen : tyUIBtn;
		tyBtnMag3PresentSen : tyUIBtn;
		tyBtnMag4PresentSen : tyUIBtn;
		tyBtnMag1ConvEntrySen : tyUIBtn;
		tyBtnMag2ConvEntrySen : tyUIBtn;
		tyBtnMag3ConvEntrySen : tyUIBtn;
		tyBtnMag4ConvEntrySen : tyUIBtn;
		tyBtnMag1AIVInPosSen1 : tyUIBtn;
		tyBtnMag1AIVInPosSen2 : tyUIBtn;
		tyBtnMag2AIVInPosSen1 : tyUIBtn;
		tyBtnMag2AIVInPosSen2 : tyUIBtn;
		tyBtnMag3AIVInPosSen1 : tyUIBtn;
		tyBtnMag3AIVInPosSen2 : tyUIBtn;
		tyBtnMag4AIVInPosSen1 : tyUIBtn;
		tyBtnMag4AIVInPosSen2 : tyUIBtn;
		tyBtnMag1OrientationChkSen1 : tyUIBtn;
		tyBtnMag2OrientationChkSen1 : tyUIBtn;
		tyBtnMag3OrientationChkSen1 : tyUIBtn;
		tyBtnMag4OrientationChkSen1 : tyUIBtn;
		tyBtnMag1OrientationChkSen2 : tyUIBtn;
		tyBtnMag2OrientationChkSen2 : tyUIBtn;
		tyBtnMag3OrientationChkSen2 : tyUIBtn;
		tyBtnMag4OrientationChkSen2 : tyUIBtn;
		tyLyr : tyUILyr;
		tyBtnMag3FixedClampCtrl : tyUIBtn;
		tyBtnMag3RemoteClampCtrl : tyUIBtn;
		tyBtnMag3ConvMtrIn : tyUIBtn;
		tyBtnMag3ConvMtrOut : tyUIBtn;
		tyBtnMag4FixedClampCtrl : tyUIBtn;
		tyBtnMag4RemoteClampCtrl : tyUIBtn;
		tyBtnMag4ConvMtrIn : tyUIBtn;
		tyBtnMag4ConvMtrOut : tyUIBtn;
		tyBtnSelUnclampRS : tyUIBtn;
		tyBtnHeightSen : tyUIBtn;
		tyBtnCAB717Sen : tyUIBtn;
		tyBtnMagSmallSen : tyUIBtn;
		tyBtnMagLargeSen : tyUIBtn;
		tyBtnMagSelClampCtrl : tyUIBtn;
	END_STRUCT;
	tyLyrP0206BypsInitConv : 	STRUCT
		tyBtnBypsInitConv : tyUIBtn;
		tyHotspotClose : tyUIHotspot;
		tyLyr : tyUILyr;
	END_STRUCT;
	tyLyrP0206OpsParam : 	STRUCT
		tyDrpDnMcMode : tyUIDrpDn;
		tyNumMinSlt : tyUINum;
		tyNumMaxSlt : tyUINum;
		tyNumPitch : tyUINum;
		tyBtnToptoBtm : tyUIBtn;
		tyNumMinSltRear : tyUINum;
		tyNumMaxSltRear : tyUINum;
		tyNumPitchRear : tyUINum;
		tyBtnToptoBtmRear : tyUIBtn;
		tyBtnSave : tyUIBtn;
		tyBtnCancel : tyUIBtn;
		tyLyr : tyUILyr;
	END_STRUCT;
END_TYPE

(**)

TYPE
	tyLyrP0300McInfo : 	STRUCT
		tyStringMcNm : tyUIString;
		tyStringJobNo : tyUIString;
		tyTxtNtAddr : tyUITxt;
		tyStringSoftwareVer : tyUIString;
		tyLyr : tyUILyr;
	END_STRUCT;
END_TYPE

(**)

TYPE
	tyLyrP0400ProdSel : 	STRUCT
		tyHotspotShowLRcp : tyUIHotspot;
		tyStringRecipeNm : tyUILString;
		tyNumProdWidth2 : tyUINum;
		tyNumProdWidth : tyUINum;
		tyNumMinSlt : tyUINum;
		tyNumMaxSlt : tyUINum;
		tyNumPitch : tyUINum;
		tyBtnToptoBtm : tyUIBtn;
		tyBtnLongBrd : tyUIBtn;
		tyBtnPreview : tyUIBtn;
		tyTableRecipe : tyUITable;
		tyStringSearch : tyUILString;
		tyBtnLoad : tyUIBtn;
		tyTxtMcMode : tyUITxt;
		tyTxtFlippedBrd : tyUITxt;
		tyBtnSort : tyUIBtn;
		tyNotQuadrupleLyr : tyUILyr;
		tyQuadrupleLyr : tyUILyr;
		tyNumMinSltRear : tyUINum;
		tyNumMaxSltRear : tyUINum;
		tyNumPitchRear : tyUINum;
		tyNumProdWidthRear : tyUINum;
		tyNumMtrPshrExtSpd : tyUINum;
		tyNumMtrPshrExtTorq : tyUINum;
		tyTxtMtrPshrExtSpd : tyUITxt;
		tyTxtMtrPshrExtTorq : tyUITxt;
		tyNumPshrOffset : tyUINum;
		tyTxtPshrOffset : tyUITxt;
	END_STRUCT;
	tyLyrP0400RcpDet : 	STRUCT
		tyHotspotShowLRcp : tyUIHotspot;
		tyStringRecipeNm : tyUILString;
		tyNumRecipeNum : tyUINum;
		tyNumProdWidth : tyUINum;
		tyNumProdWidth2 : tyUINum;
		tyNumProdWidthRear : tyUINum;
		tyNumFirstSlt : tyUINum;
		tyNumLastSlt : tyUINum;
		tyNumPitch : tyUINum;
		tyBtnToptoBtm : tyUIBtn;
		tyBtnLongBrd : tyUIBtn;
		tyTxtMcMode : tyUITxt;
		tyTxtFlippedBrd : tyUITxt;
		tyHotspotClose : tyUIHotspot;
		tyLyr : tyUILyr;
		tyLyr1 : tyUILyr;
		tyNumMtrPshrExtSpd : tyUINum;
		tyNumMtrPshrExtTorq : tyUINum;
		tyTxtMtrPshrExtSpd : tyUITxt;
		tyTxtMtrPshrExtTorq : tyUITxt;
		tyNumPshrOffset : tyUINum;
		tyTxtPshrOffset : tyUITxt;
	END_STRUCT;
END_TYPE

(**)

TYPE
	tyLyrP0410MagSel : 	STRUCT
		tyStringRecipeNm : tyUIString;
		tyNumSltToSltDist : tyUINum;
		tyNumMaxSlt : tyUINum;
		tyNumLifterMag1Slt1Pos : tyUINum;
		tyNumLifterMag2Slt1Pos : tyUINum;
		tyNumLifterMag3Slt1Pos : tyUINum;
		tyNumLifterMag4Slt1Pos : tyUINum;
		tyNumTravPosMag1 : tyUINum;
		tyNumTravPosMag2 : tyUINum;
		tyNumTravPosMag3 : tyUINum;
		tyNumTravPosMag4 : tyUINum;
		tyTxtLifMag3Slt1PosLbl : tyUITxt;
		tyTxtTravPosMag3Lbl : tyUITxt;
		tyBtnLoad : tyUIBtn;
		tyBtnPreview : tyUIBtn;
		tyTableRecipe : tyUITable;
		tyTxtMagModel : tyUITxt;
		tyNumMagMaxBrdWidth : tyUINum;
		tyTxtMagTitle : tyUITxt;
		tyBtnSort : tyUIBtn;
		tyBtnSafetyBar : tyUIBtn;
		tyBtnMagHeightChkEn : tyUIBtn;
		tyBitmapBrder : tyUIBitmap;
	END_STRUCT;
	tyLyrP0410MagDet : 	STRUCT
		tyStringRecipeNm : tyUIString;
		tyNumSltToSltDist : tyUINum;
		tyNumMaxSlt : tyUINum;
		tyNumLifterMag1Slt1Pos : tyUINum;
		tyNumLifterMag2Slt1Pos : tyUINum;
		tyNumLifterMag3Slt1Pos : tyUINum;
		tyNumLifterMag4Slt1Pos : tyUINum;
		tyNumTravPosMag1 : tyUINum;
		tyNumTravPosMag2 : tyUINum;
		tyNumTravPosMag3 : tyUINum;
		tyNumTravPosMag4 : tyUINum;
		tyTxtLifMag3Slt1PosLbl : tyUITxt;
		tyTxtTravPosMag3Lbl : tyUITxt;
		tyTxtMagModel : tyUITxt;
		tyHotspotClose : tyUIHotspot;
		tyNumMagMaxBrdWidth : tyUINum;
		tyLyr : tyUILyr;
		tyBtnSafetyBar : tyUIBtn;
		tyBtnMagHeightChkEn : tyUIBtn;
	END_STRUCT;
END_TYPE

(**)

TYPE
	tyLyrP0600Alm : 	STRUCT
		tyBtnCurr : tyUIBtn;
		tyBtnHistory : tyUIBtn;
		a_tyStringAlm : ARRAY[1..c_uiP0600TableSize]OF tyUILString;
		a_tyHotspotAlm : ARRAY[1..c_uiP0600TableSize]OF tyUIHotspot;
		tyLyr : tyUILyr;
		tyAlarm : tyUIAlarm;
		tyBtnHistoryUp : tyUIBtn;
		tyBtnHistoryDown : tyUIBtn;
	END_STRUCT;
END_TYPE

(**)

TYPE
	tyLyrP0700LFCtrl : 	STRUCT
		tyBtnChgAll : tyUIBtn;
		tyBtnChgSeqAuto : tyUIBtn;
		tyBtnChgSeqMnl : tyUIBtn;
		tyBtnSyncTm : tyUIBtn;
		tyBitmapChgAll : tyUIBitmap;
		tyBitmapChgSeqAuto : tyUIBitmap;
		tyBitmapChgSeqMnl : tyUIBitmap;
		tyBitmapSyncTm : tyUIBitmap;
		tyTable1List : tyUITable1;
		tyLyr : tyUILyr;
	END_STRUCT;
END_TYPE

(**)

TYPE
	tyLyrP0800MagInfo1 : 	STRUCT
		tyTable1List : tyUITable1;
		tyTable2List : tyUITable1;
		tyTxtMag1Stat : tyUITxt;
		tyTxtMag2Stat : tyUITxt;
		tyBtnMag1SetEmpty : tyUIBtn;
		tyBtnMag2SetEmpty : tyUIBtn;
		tyLyr : tyUILyr;
	END_STRUCT;
	tyLyrP0800MagInfo2 : 	STRUCT
		tyTable3List : tyUITable1;
		tyTxtMag3Stat : tyUITxt;
		tyBtnMag3SetEmpty : tyUIBtn;
		tyLyr : tyUILyr;
	END_STRUCT;
	tyLyrP0800MagInfo3 : 	STRUCT
		tyTable4List : tyUITable1;
		tyTxtMag4Stat : tyUITxt;
		tyBtnMag4SetEmpty : tyUIBtn;
		tyLyr : tyUILyr;
	END_STRUCT;
END_TYPE

(**)

TYPE
	tyLyrP0900GenIn1 : 	STRUCT
		tyBtnEStop : tyUIBtn;
		tyBtnCoverSW : tyUIBtn;
		tyBtnSafetyRly : tyUIBtn;
		tyBtnCurtainSafetyRly : tyUIBtn;
		tyBtnLifterTimingBeltSen : tyUIBtn;
		tyBtnLifterSafetyLmtSW1 : tyUIBtn;
		tyBtnLifterSafetyLmtSW2 : tyUIBtn;
		tyBtnMag1PresentSen : tyUIBtn;
		tyBtnMag2PresentSen : tyUIBtn;
		tyBtnMag3PresentSen : tyUIBtn;
		tyBtnMag4PresentSen : tyUIBtn;
		tyBtnMagWidthChk : tyUIBtn;
	END_STRUCT;
	tyLyrP0900GenIn2 : 	STRUCT
		tyBtnMag1OrientationChkSen1 : tyUIBtn;
		tyBtnMag2OrientationChkSen1 : tyUIBtn;
		tyBtnMag3OrientationChkSen1 : tyUIBtn;
		tyBtnMag4OrientationChkSen1 : tyUIBtn;
		tyBtnMag1OrientationChkSen2 : tyUIBtn;
		tyBtnMag2OrientationChkSen2 : tyUIBtn;
		tyBtnMag3OrientationChkSen2 : tyUIBtn;
		tyBtnMag4OrientationChkSen2 : tyUIBtn;
		tyLyr : tyUILyr;
	END_STRUCT;
END_TYPE

(**)

TYPE
	tyLyrP0910GenOut : 	STRUCT
		tyBtnTLGreen : tyUIBtn;
		tyBtnTLRed : tyUIBtn;
		tyBtnTLAmber : tyUIBtn;
		tyBtnBuzzer : tyUIBtn;
		tyBtnSafetyCurtainRst : tyUIBtn; (*moved to new layer*)
		tyBtnCurtainByp : tyUIBtn;
		tyBtnCurtainPBLED : tyUIBtn;
		tyBtnSafetyRst : tyUIBtn;
	END_STRUCT;
	tyLyrP0910GenOutCurtainSen : 	STRUCT
		tyBtnBypCurtainSenPBLED : tyUIBtn;
		tyBtnBypCurtainSen : tyUIBtn;
		tyBtnRstCurtainSen : tyUIBtn;
		tyLyr : tyUILyr;
	END_STRUCT;
END_TYPE

(**)

TYPE
	tyLyrP0920MtrNPneuCtrl : 	STRUCT
		tyBtnAW : tyUIBtn;
		tyBtnAWPushPul : tyUIBtn;
		tyBtnTrav : tyUIBtn;
		tyBtnLifter : tyUIBtn;
		tyBtnPullerConv : tyUIBtn;
		tyBtnMag1Conv : tyUIBtn;
		tyBtnMag2Conv : tyUIBtn;
		tyBtnMag3Conv : tyUIBtn;
		tyLyr : tyUILyr;
	END_STRUCT;
	tyLyrP0920MtrNPneuCtrlPneu : 	STRUCT
		tyBtnShutter : tyUIBtn;
		tyBtnSafetyBar : tyUIBtn;
		tyBtnTrolleyLck : tyUIBtn;
		tyLyr : tyUILyr;
	END_STRUCT;
END_TYPE

(**)

TYPE
	tyLyrP0921InletShutterCom : 	STRUCT
		tyBtnSwitch : tyUIBtn;
		tyBitmapMc : tyUIBitmap;
		tyBtnOpenRS : tyUIBtn;
		tyBtnCloseRS : tyUIBtn;
		tyTxtTit : tyUITxt;
		tyLyr : tyUILyr;
	END_STRUCT;
	tyLyrP0921InletShutterDC : 	STRUCT
		tyBtnOpen : tyUIBtn;
		tyBtnOpen2 : tyUIBtn;
		tyBtnOpen3 : tyUIBtn;
		tyBtnClose : tyUIBtn;
		tyLyr : tyUILyr;
	END_STRUCT;
	tyLyrP0921InletShutterFB : 	STRUCT
		tyStringStat : tyUILString;
		tyBtnOpen : tyUIBtn;
		tyBtnClose : tyUIBtn;
		tyBtnOpen2 : tyUIBtn;
		tyBtnOpen3 : tyUIBtn;
		tyBtnOpenRS2 : tyUIBtn;
		tyBtnOpenRS3 : tyUIBtn;
		tyBtnCloseRS2 : tyUIBtn;
		tyBtnCloseRS3 : tyUIBtn;
		tyLyr : tyUILyr;
	END_STRUCT;
	tyLyrP0921OutletShutterCom : 	STRUCT
		tyBtnSwitch : tyUIBtn;
		tyBitmapMc : tyUIBitmap;
		tyBtnOpenRS : tyUIBtn;
		tyBtnCloseRS : tyUIBtn;
		tyTxtTit : tyUITxt;
		tyLyr : tyUILyr;
	END_STRUCT;
	tyLyrP0921OutletShutterDC : 	STRUCT
		tyBtnOpen : tyUIBtn;
		tyBtnClose : tyUIBtn;
		tyLyr : tyUILyr;
	END_STRUCT;
	tyLyrP0921OutletShutterFB : 	STRUCT
		tyStringStat : tyUILString;
		tyBtnOpen : tyUIBtn;
		tyBtnClose : tyUIBtn;
		tyBtnOpen2 : tyUIBtn;
		tyBtnOpen3 : tyUIBtn;
		tyBtnOpenRS2 : tyUIBtn;
		tyBtnOpenRS3 : tyUIBtn;
		tyBtnCloseRS2 : tyUIBtn;
		tyBtnCloseRS3 : tyUIBtn;
		tyLyr : tyUILyr;
	END_STRUCT;
	tyLyrP0921OutletShutterDis : 	STRUCT
		tyLyr : tyUILyr;
	END_STRUCT;
END_TYPE

(**)

TYPE
	tyLyrP0923LftSafetyBarCom : 	STRUCT
		tyBitmapMc : tyUIBitmap;
		tyBtnSwitch : tyUIBtn;
		tyBtnExtRS : tyUIBtn;
		tyBtnRetRS : tyUIBtn;
		tyTxtSubTitle : tyUITxt;
		tyLyr : tyUILyr;
	END_STRUCT;
	tyLyrP0923LftSafetyBarDC : 	STRUCT
		tyBtnExt : tyUIBtn;
		tyBtnRet : tyUIBtn;
		tyLyr : tyUILyr;
	END_STRUCT;
	tyLyrP0923LftSafetyBarFB : 	STRUCT
		tyStringStat : tyUILString;
		tyBtnExt : tyUIBtn;
		tyBtnRet : tyUIBtn;
		tyLyr : tyUILyr;
	END_STRUCT;
	tyLyrP0923RgtSafetyBarCom : 	STRUCT
		tyBitmapMc : tyUIBitmap;
		tyBtnSwitch : tyUIBtn;
		tyBtnExtRS : tyUIBtn;
		tyBtnRetRS : tyUIBtn;
		tyTxtSubTitle : tyUITxt;
		tyLyr : tyUILyr;
	END_STRUCT;
	tyLyrP0923RgtSafetyBarDC : 	STRUCT
		tyBtnExt : tyUIBtn;
		tyBtnRet : tyUIBtn;
		tyLyr : tyUILyr;
	END_STRUCT;
	tyLyrP0923RgtSafetyBarFB : 	STRUCT
		tyStringStat : tyUILString;
		tyBtnExt : tyUIBtn;
		tyBtnRet : tyUIBtn;
		tyLyr : tyUILyr;
	END_STRUCT;
END_TYPE

(**)

TYPE
	tyLyrP0924TrolleyLckCom : 	STRUCT
		tyBitmapMc : tyUIBitmap;
		tyBtnSwitch : tyUIBtn;
		tyBtnExtRS : tyUIBtn;
		tyBtnExtRS2 : tyUIBtn;
		tyBtnPresentSen1 : tyUIBtn;
		tyBtnPresentSen2 : tyUIBtn;
		tyTxtSubTitle : tyUITxt;
		tyLyr : tyUILyr;
	END_STRUCT;
	tyLyrP0924TrolleyLckDC : 	STRUCT
		tyBtnExt : tyUIBtn;
		tyBtnRet : tyUIBtn;
		tyBtnExt2 : tyUIBtn;
		tyBtnRet2 : tyUIBtn;
		tyLyr : tyUILyr;
	END_STRUCT;
	tyLyrP0924TrolleyLckFB : 	STRUCT
		tyStringStat : tyUILString;
		tyBtnExt : tyUIBtn;
		tyBtnRet : tyUIBtn;
		tyBtnExt2 : tyUIBtn;
		tyBtnRet2 : tyUIBtn;
		tyLyr : tyUILyr;
	END_STRUCT;
END_TYPE

(**)

TYPE
	tyLyrP0930Mag1ConvCom : 	STRUCT
		tyBitmapMc : tyUIBitmap;
		tyBtnSwitch : tyUIBtn;
		tyBtnMagPresentSen : tyUIBtn;
		tyBtnMagOrientationChkSen1 : tyUIBtn;
		tyBtnMagOrientationChkSen2 : tyUIBtn;
		tyBtnMagConvEntSen : tyUIBtn;
		tyBtnMagAIVPosSen1 : tyUIBtn;
		tyBtnMagAIVPosSen2 : tyUIBtn;
		tyBtnSelClampRS : tyUIBtn;
		tyBtnSelUnclampRS : tyUIBtn;
		tyBtnFixedClampRS : tyUIBtn;
		tyBtnFixedUnclampRS : tyUIBtn;
		tyBtnRemoteClampRS : tyUIBtn;
		tyBtnRemoteUnclampRS : tyUIBtn;
		tyBtnHeightSen : tyUIBtn;
		tyBtnCAB717Sen : tyUIBtn;
		tyBtnMagSmallSen : tyUIBtn;
		tyBtnMagLargeSen : tyUIBtn;
		tyLyr : tyUILyr;
		tyBtnMagDetSen : tyUIBtn;
		tyBtnSltLckSen : tyUIBtn;
	END_STRUCT;
	tyLyrP0930Mag1ConvDC : 	STRUCT
		tyBtnMagIn : tyUIBtn;
		tyBtnMagOut : tyUIBtn;
		tyBtnStop : tyUIBtn;
		tyBtnSelClamp : tyUIBtn;
		tyBtnSelUnclamp : tyUIBtn;
		tyBtnFixedClamp : tyUIBtn;
		tyBtnFixedUnclamp : tyUIBtn;
		tyBtnRemoteClamp : tyUIBtn;
		tyBtnRemoteUnclamp : tyUIBtn;
		tyLyr : tyUILyr;
		tyLyrWithoutSelClamp : tyUILyr;
	END_STRUCT;
	tyLyrP0930Mag1ConvFB : 	STRUCT
		tyStringStat : tyUILString;
		tyBtnEnt : tyUIBtn;
		tyBtnExit : tyUIBtn;
		tyBtnStop : tyUIBtn;
		tyBtnSelClamp : tyUIBtn;
		tyBtnSelUnclamp : tyUIBtn;
		tyBtnFixedClamp : tyUIBtn;
		tyBtnFixedUnclamp : tyUIBtn;
		tyBtnRemoteClamp : tyUIBtn;
		tyBtnRemoteUnclamp : tyUIBtn;
		tyLyr : tyUILyr;
		tyLyrWithoutSelClamp : tyUILyr;
	END_STRUCT;
END_TYPE

(**)

TYPE
	tyLyrP0931Mag2ConvCom : 	STRUCT
		tyBitmapMc : tyUIBitmap;
		tyBtnSwitch : tyUIBtn;
		tyBtnMagPresentSen : tyUIBtn;
		tyBtnMagOrientationChkSen1 : tyUIBtn;
		tyBtnMagOrientationChkSen2 : tyUIBtn;
		tyBtnMagConvEntSen : tyUIBtn;
		tyBtnMagAIVPosSen1 : tyUIBtn;
		tyBtnMagAIVPosSen2 : tyUIBtn;
		tyBtnSelClampRS : tyUIBtn;
		tyBtnSelUnclampRS : tyUIBtn;
		tyBtnFixedClampRS : tyUIBtn;
		tyBtnFixedUnclampRS : tyUIBtn;
		tyBtnRemoteClampRS : tyUIBtn;
		tyBtnRemoteUnclampRS : tyUIBtn;
		tyBtnHeightSen : tyUIBtn;
		tyBtnCAB717Sen : tyUIBtn;
		tyBtnMagSmallSen : tyUIBtn;
		tyBtnMagLargeSen : tyUIBtn;
		tyLyr : tyUILyr;
		tyBtnMagDetSen : tyUIBtn;
		tyBtnSltLckSen : tyUIBtn;
	END_STRUCT;
	tyLyrP0931Mag2ConvDC : 	STRUCT
		tyBtnMagIn : tyUIBtn;
		tyBtnMagOut : tyUIBtn;
		tyBtnStop : tyUIBtn;
		tyBtnSelClamp : tyUIBtn;
		tyBtnSelUnclamp : tyUIBtn;
		tyBtnFixedClamp : tyUIBtn;
		tyBtnFixedUnclamp : tyUIBtn;
		tyBtnRemoteClamp : tyUIBtn;
		tyBtnRemoteUnclamp : tyUIBtn;
		tyLyr : tyUILyr;
		tyLyrWithoutSelClamp : tyUILyr;
	END_STRUCT;
	tyLyrP0931Mag2ConvFB : 	STRUCT
		tyStringStat : tyUILString;
		tyBtnEnt : tyUIBtn;
		tyBtnExit : tyUIBtn;
		tyBtnStop : tyUIBtn;
		tyBtnSelClamp : tyUIBtn;
		tyBtnSelUnclamp : tyUIBtn;
		tyBtnFixedClamp : tyUIBtn;
		tyBtnFixedUnclamp : tyUIBtn;
		tyBtnRemoteClamp : tyUIBtn;
		tyBtnRemoteUnclamp : tyUIBtn;
		tyLyr : tyUILyr;
		tyLyrWithoutSelClamp : tyUILyr;
	END_STRUCT;
END_TYPE

(**)

TYPE
	tyLyrP0932Mag3ConvCom : 	STRUCT
		tyBitmapMc : tyUIBitmap;
		tyBtnSwitch : tyUIBtn;
		tyBtnMagPresentSen : tyUIBtn;
		tyBtnMagOrientationChkSen1 : tyUIBtn;
		tyBtnMagOrientationChkSen2 : tyUIBtn;
		tyBtnMagConvEntSen : tyUIBtn;
		tyBtnMagAIVPosSen1 : tyUIBtn;
		tyBtnMagAIVPosSen2 : tyUIBtn;
		tyBtnSelClampRS : tyUIBtn;
		tyBtnSelUnclampRS : tyUIBtn;
		tyBtnFixedClampRS : tyUIBtn;
		tyBtnFixedUnclampRS : tyUIBtn;
		tyBtnRemoteClampRS : tyUIBtn;
		tyBtnRemoteUnclampRS : tyUIBtn;
		tyBtnHeightSen : tyUIBtn;
		tyBtnCAB717Sen : tyUIBtn;
		tyBtnMagSmallSen : tyUIBtn;
		tyBtnMagLargeSen : tyUIBtn;
		tyLyr : tyUILyr;
		tyBtnMagDetSen : tyUIBtn;
	END_STRUCT;
	tyLyrP0932Mag3ConvDC : 	STRUCT
		tyBtnMagIn : tyUIBtn;
		tyBtnMagOut : tyUIBtn;
		tyBtnStop : tyUIBtn;
		tyBtnSelClamp : tyUIBtn;
		tyBtnSelUnclamp : tyUIBtn;
		tyBtnFixedClamp : tyUIBtn;
		tyBtnFixedUnclamp : tyUIBtn;
		tyBtnRemoteClamp : tyUIBtn;
		tyBtnRemoteUnclamp : tyUIBtn;
		tyLyr : tyUILyr;
		tyLyrWithoutSelClamp : tyUILyr;
	END_STRUCT;
	tyLyrP0932Mag3ConvFB : 	STRUCT
		tyStringStat : tyUILString;
		tyBtnEnt : tyUIBtn;
		tyBtnExit : tyUIBtn;
		tyBtnStop : tyUIBtn;
		tyBtnSelClamp : tyUIBtn;
		tyBtnSelUnclamp : tyUIBtn;
		tyBtnFixedClamp : tyUIBtn;
		tyBtnFixedUnclamp : tyUIBtn;
		tyBtnRemoteClamp : tyUIBtn;
		tyBtnRemoteUnclamp : tyUIBtn;
		tyLyr : tyUILyr;
		tyLyrWithoutSelClamp : tyUILyr;
	END_STRUCT;
END_TYPE

(**)

TYPE
	tyLyrP0939Mag4ConvCom : 	STRUCT
		tyBitmapMc : tyUIBitmap;
		tyBtnSwitch : tyUIBtn;
		tyBtnMagPresentSen : tyUIBtn;
		tyBtnMagOrientationChkSen1 : tyUIBtn;
		tyBtnMagOrientationChkSen2 : tyUIBtn;
		tyBtnMagConvEntSen : tyUIBtn;
		tyBtnMagAIVPosSen1 : tyUIBtn;
		tyBtnMagAIVPosSen2 : tyUIBtn;
		tyBtnSelClampRS : tyUIBtn;
		tyBtnSelUnclampRS : tyUIBtn;
		tyBtnFixedClampRS : tyUIBtn;
		tyBtnFixedUnclampRS : tyUIBtn;
		tyBtnRemoteClampRS : tyUIBtn;
		tyBtnRemoteUnclampRS : tyUIBtn;
		tyBtnHeightSen : tyUIBtn;
		tyBtnCAB717Sen : tyUIBtn;
		tyBtnMagSmallSen : tyUIBtn;
		tyBtnMagLargeSen : tyUIBtn;
		tyLyr : tyUILyr;
	END_STRUCT;
	tyLyrP0939Mag4ConvDC : 	STRUCT
		tyBtnMagIn : tyUIBtn;
		tyBtnMagOut : tyUIBtn;
		tyBtnStop : tyUIBtn;
		tyBtnSelClamp : tyUIBtn;
		tyBtnSelUnclamp : tyUIBtn;
		tyBtnFixedClamp : tyUIBtn;
		tyBtnFixedUnclamp : tyUIBtn;
		tyBtnRemoteClamp : tyUIBtn;
		tyBtnRemoteUnclamp : tyUIBtn;
		tyLyr : tyUILyr;
		tyLyrWithoutSelClamp : tyUILyr;
	END_STRUCT;
	tyLyrP0939Mag4ConvFB : 	STRUCT
		tyStringStat : tyUILString;
		tyBtnEnt : tyUIBtn;
		tyBtnExit : tyUIBtn;
		tyBtnStop : tyUIBtn;
		tyBtnSelClamp : tyUIBtn;
		tyBtnSelUnclamp : tyUIBtn;
		tyBtnFixedClamp : tyUIBtn;
		tyBtnFixedUnclamp : tyUIBtn;
		tyBtnRemoteClamp : tyUIBtn;
		tyBtnRemoteUnclamp : tyUIBtn;
		tyLyr : tyUILyr;
		tyLyrWithoutSelClamp : tyUILyr;
	END_STRUCT;
END_TYPE

(**)

TYPE
	tyLyrP0933PullConvCom : 	STRUCT
		tyBitmapMc : tyUIBitmap;
		tyBtnSwitch : tyUIBtn;
		tyBtnLftSen : tyUIBtn;
		tyBtnRgtSen : tyUIBtn;
		tyBtnExtRS : tyUIBtn;
		tyBtnRetRS : tyUIBtn;
		tyBtnRotHmRS : tyUIBtn;
		tyBtnRotRmRS : tyUIBtn;
		tyBtnAlarmSig : tyUIBtn;
		tyBtnTorqueSig : tyUIBtn;
		tyBtnExtSen : tyUIBtn;
		tyBtnExtSlwSen : tyUIBtn;
		tyBtnRetSen : tyUIBtn;
		tyBtnRetSlwSen : tyUIBtn;
		tyBtnAntiJamSen : tyUIBtn;
		tyLyr : tyUILyr;
		tyBtnConvClrSen : tyUIBtn;
	END_STRUCT;
	tyLyrP0933PullConvDC : 	STRUCT
		tyBtnStart : tyUIBtn;
		tyBtnStop : tyUIBtn;
		tyBtnExt : tyUIBtn;
		tyBtnRet : tyUIBtn;
		tyBtnRotToHm : tyUIBtn;
		tyBtnRotToRm : tyUIBtn;
		tyBtnSpdBinBit0 : tyUIBtn;
		tyBtnSpdBinBit1 : tyUIBtn;
		tyBtnSpdBinBit2 : tyUIBtn;
		tyBtnSigOn : tyUIBtn;
		tyBtnBrake : tyUIBtn;
		tyBtnAlarmRst : tyUIBtn;
		tyLyr : tyUILyr;
	END_STRUCT;
	tyLyrP0933PullConvFB : 	STRUCT
		tyStringStat : tyUILString;
		tyBtnEnt : tyUIBtn;
		tyBtnExit : tyUIBtn;
		tyBtnCylEnt : tyUIBtn;
		tyBtnStop : tyUIBtn;
		tyBtnExt : tyUIBtn;
		tyBtnRet : tyUIBtn;
		tyBtnRotToHm : tyUIBtn;
		tyBtnRotToRm : tyUIBtn;
		tyNumExtSpd : tyUINum;
		tyNumExtTorqPercent : tyUINum;
		tyLyr : tyUILyr;
	END_STRUCT;
END_TYPE

(**)

TYPE
	tyLyrP0934AW : 	STRUCT
		tyNumNewWidth : tyUINum;
		tyBtnGo : tyUIBtn;
	END_STRUCT;
END_TYPE

(**)

TYPE
	tyLyrP0935Lifter : 	STRUCT
		tyNumNewSlt : tyUINum;
		tyBtnGo : tyUIBtn;
		tyBtnGoLaneA : tyUIBtn;
		tyBtnGoLaneB : tyUIBtn;
		tyBtnNxtSlt : tyUIBtn;
		tyBtnPrevSlt : tyUIBtn;
		tyNumMagPos : tyUINum;
	END_STRUCT;
END_TYPE

(**)

TYPE
	tyLyrP0936Trav : 	STRUCT
		tyBtnGoToLaneA : tyUIBtn;
		tyBtnGoToLaneB : tyUIBtn;
		tyBtnGoToMag1 : tyUIBtn;
		tyBtnGoToMag2 : tyUIBtn;
		tyBtnGoToMag3 : tyUIBtn;
		tyBtnGoToMag4 : tyUIBtn;
	END_STRUCT;
END_TYPE

(**)

TYPE
	tyLyrP0937AWPushOrPuller : 	STRUCT
		tyNumNewWidth : tyUINum;
		tyBtnGo : tyUIBtn;
	END_STRUCT;
	tyLyrP0937InOutletShutterFB : 	STRUCT
		tyStringStat : tyUILString;
		tyBtnOpen : tyUIBtn;
		tyBtnClose : tyUIBtn;
		tyLyr : tyUILyr;
	END_STRUCT;
END_TYPE

(**)

TYPE
	tyLyrP0940CommCtrlDSSMEMA : 	STRUCT
		tyBtnDSB : tyUIBtn;
		tyBtnDBA : tyUIBtn;
		tyLyr : tyUILyr;
	END_STRUCT;
	tyLyrP0940SOTComm : 	STRUCT
		tyBtnAIVRcv1 : tyUIBtn;
		tyBtnAIVErr1 : tyUIBtn;
		tyBtnAIVRdy1 : tyUIBtn;
		tyBtnAIVAvail1 : tyUIBtn;
		tyBtnAIVSLarge1 : tyUIBtn;
		tyBtnMagErr1 : tyUIBtn;
		tyBtnMagRdy1 : tyUIBtn;
		tyBtnMagAvail1 : tyUIBtn;
		tyBtnMagSLarge1 : tyUIBtn;
		tyBtnAIVRcv2 : tyUIBtn;
		tyBtnAIVErr2 : tyUIBtn;
		tyBtnAIVRdy2 : tyUIBtn;
		tyBtnAIVAvail2 : tyUIBtn;
		tyBtnAIVSLarge2 : tyUIBtn;
		tyBtnMagErr2 : tyUIBtn;
		tyBtnMagRdy2 : tyUIBtn;
		tyBtnMagAvail2 : tyUIBtn;
		tyBtnMagSLarge2 : tyUIBtn;
		tyBtnAIVRcv3 : tyUIBtn;
		tyBtnAIVErr3 : tyUIBtn;
		tyBtnAIVRdy3 : tyUIBtn;
		tyBtnAIVAvail3 : tyUIBtn;
		tyBtnAIVSLarge3 : tyUIBtn;
		tyBtnMagErr3 : tyUIBtn;
		tyBtnMagRdy3 : tyUIBtn;
		tyBtnMagAvail3 : tyUIBtn;
		tyBtnMagSLarge3 : tyUIBtn;
		tyBtnAIVRcv4 : tyUIBtn;
		tyBtnAIVErr4 : tyUIBtn;
		tyBtnAIVRdy4 : tyUIBtn;
		tyBtnAIVAvail4 : tyUIBtn;
		tyBtnAIVSLarge4 : tyUIBtn;
		tyBtnMagErr4 : tyUIBtn;
		tyBtnMagRdy4 : tyUIBtn;
		tyBtnMagAvail4 : tyUIBtn;
		tyBtnMagSLarge4 : tyUIBtn;
		tyBtnFleetMgrActive : tyUIBtn;
		tyBtnMagReqBring1 : tyUIBtn;
		tyBtnMagReqtGet1 : tyUIBtn;
		tyBtnMagReqBring2 : tyUIBtn;
		tyBtnMagReqtGet2 : tyUIBtn;
		tyBtnMagReqBring3 : tyUIBtn;
		tyBtnMagReqtGet3 : tyUIBtn;
		tyBtnMagReqBring4 : tyUIBtn;
		tyBtnMagReqtGet4 : tyUIBtn;
		tySOTLyr1 : tyUILyr;
		tySOTLyr2 : tyUILyr;
		tySOTLyr3 : tyUILyr;
		tySOTLyr4 : tyUILyr;
		tyTxtAIVCommProtocol : tyUITxt;
	END_STRUCT;
END_TYPE

(**)

TYPE
	tyLyrP0950Simu : 	STRUCT
		tyBtnSimu : tyUIBtn;
		tyBtnStart : tyUIBtn;
		tyBtnStop : tyUIBtn;
		tyBtnSOT1 : tyLyrP0950SOTBtn;
		tyBtnSOT2 : tyLyrP0950SOTBtn;
		tyBtnSOT3 : tyLyrP0950SOTBtn;
		tyBtnSOT4 : tyLyrP0950SOTBtn;
		tyBtnMagSOT1 : tyLyrP0950SOTBtn;
		tyBtnMagSOT2 : tyLyrP0950SOTBtn;
		tyBtnMagSOT3 : tyLyrP0950SOTBtn;
		tyBtnMagSOT4 : tyLyrP0950SOTBtn;
		tyBtnInShutterSim : tyUIBtn;
		tyBtnTestTrav : tyUIBtn;
		tyBtnNtParaWr : tyUIBtn;
		tyBtnNtParaWr2 : tyUIBtn;
		tyStringJobNo : tyUILString;
		tyNumAddr : tyUINum;
		tyNumTravSpd : tyUINum;
		tyNumLifterSpd : tyUINum;
		tyBtnRcpGen : tyUIBtn;
		tyLyrMag3 : tyUILyr;
		tyLyrMag4 : tyUILyr;
		tyLyr1 : tyUILyr;
		tyLyr : tyUILyr;
	END_STRUCT;
	tyLyrP0950SimuAGVToMC : 	STRUCT
		tyBtnAGVSimulateOn : tyUIBtn;
		tyBtnAGVOnline : tyUIBtn;
		tyBtnAGVInPos1 : tyUIBtn;
		tyBtnAGVInPos2 : tyUIBtn;
		tyBtnAGVInPos3 : tyUIBtn;
		tyBtnAGVAuto : tyUIBtn;
		tyBtnAGV1Occupied : tyUIBtn;
		tyBtnAGV2Occupied : tyUIBtn;
		tyBtnAGV3Occupied : tyUIBtn;
		tyLyr : tyUILyr;
	END_STRUCT;
	tyLyrP0950SimuMCToAGV : 	STRUCT
		tyBtnMachineOnline : tyUIBtn;
		tyBtnMachineEstop : tyUIBtn;
		tyBtnMag1Empty : tyUIBtn;
		tyBtnMag2Empty : tyUIBtn;
		tyBtnMag3Empty : tyUIBtn;
		tyBtnMag1Rdy : tyUIBtn;
		tyBtnMag2Rdy : tyUIBtn;
		tyBtnMag3Rdy : tyUIBtn;
		tyBtnMag1Auto : tyUIBtn;
		tyBtnMag2Auto : tyUIBtn;
		tyBtnMag3Auto : tyUIBtn;
		tyBtnMag1Occupied : tyUIBtn;
		tyBtnMag2Occupied : tyUIBtn;
		tyBtnMag3Occupied : tyUIBtn;
		tyBtnMag1IncorrectModel : tyUIBtn;
		tyBtnMag2IncorrectModel : tyUIBtn;
		tyBtnMag3IncorrectModel : tyUIBtn;
	END_STRUCT;
	tyLyrP0950SOTBtn : 	STRUCT
		tyBtnInPos : tyUIBtn;
		tyBtnError : tyUIBtn;
		tyBtnRdy : tyUIBtn;
		tyBtnAvail : tyUIBtn;
		tyBtnSize : tyUIBtn;
	END_STRUCT;
	tyLyrP0950SOTstatus : 	STRUCT
		tyBtnInPos : BOOL;
		tyBtnError : BOOL;
		tyBtnRdy : BOOL;
		tyBtnAvail : BOOL;
	END_STRUCT;
END_TYPE

(**)

TYPE
	tyLyrP1000Lang : 	STRUCT
		tyBtnChinese : tyUIBtn;
		tyBtnEnglish : tyUIBtn;
		tyBtnGerman : tyUIBtn;
		tyNumYear : tyUINum;
		tyNumMonth : tyUINum;
		tyNumDay : tyUINum;
		tyNumHour : tyUINum;
		tyNumMinute : tyUINum;
		tyNumSecond : tyUINum;
	END_STRUCT;
END_TYPE

(**)

TYPE
	tyLyrP1020McSetNavi : 	STRUCT
		tyBtnMcSet : tyUIBtn;
		tyBtnVCommSet : tyUIBtn;
		tyBtnHCommSet : tyUIBtn;
		tyBtnUSBSet : tyUIBtn;
		tyBtnAntiGapSet : tyUIBtn;
		tyBtnAIVCommSet : tyUIBtn;
		tyBtnRS232Set : tyUIBtn;
		tyLyr : tyUILyr;
	END_STRUCT;
END_TYPE

(**)

TYPE
	tyLyrP1021McSetGen : 	STRUCT
		tyStringMcNm : tyUIString;
		tyDrpDnDefaultMcMod : tyUIDrpDn;
		tyDrpDnDefaultFlippedBrd : tyUIDrpDn;
		tyDrpDnNetworkMod : tyUIDrpDn;
		tyNumSSaverTm : tyUINum;
		tyBtnSSaverEn : tyUIBtn;
		tyTxtLblSSaver : tyUITxt;
		tyStringIPAddr : tyUIString;
		tyStringSubnetMask : tyUIString;
		tyTxtWidthAtHm : tyUITxt;
		tyNumWidthAtHm : tyUINum;
		tyTxtAWPusherAtHm : tyUITxt;
		tyBtnAWPusherDis : tyUIBtn;
		tyNumConvInitTm : tyUINum;
		tyNumTranOutErrDlyTm : tyUINum;
		tyTxtMag1ConvRunTm : tyUITxt;
		tyNumMag1ConvRunTm : tyUINum;
		tyTxtMag2ConvRunTm : tyUITxt;
		tyNumMag2ConvRunTm : tyUINum;
		tyTxtMag3ConvRunTm : tyUITxt;
		tyNumMag3ConvRunTm : tyUINum;
		tyTxtMag4ConvRunTm : tyUITxt;
		tyNumMag4ConvRunTm : tyUINum;
		tyNumTravPosLaneA : tyUINum;
		tyNumLiftPosLaneA : tyUINum;
		tyTxtLiftPosLaneA : tyUITxt;
		tyTxtTravPosLaneB : tyUITxt;
		tyNumTravPosLaneB : tyUINum;
		tyTxtLiftPosLaneB : tyUITxt;
		tyNumLiftPosLaneB : tyUINum;
		tyBtnTravPosATeach : tyUIBtn;
		tyBtnTravPosBTeach : tyUIBtn;
		tyBtnLiftPosATeach : tyUIBtn;
		tyBtnLiftPosBTeach : tyUIBtn;
		tyBtnAWDis : tyUIBtn;
		tyBtnMnlAccDat : tyUIBtn;
		tyBtnAutoStepEn : tyUIBtn;
		tyBtnVSMEMAEn : tyUIBtn;
		tyBtnHermesRmtEn : tyUIBtn;
		tyBtnLongBrdEn : tyUIBtn;
		tyBtnOutShutterDis : tyUIBtn;
		tyBtnChgParamEn : tyUIBtn;
		tyLyrGen1 : tyUILyr;
		tyLyrGen2 : tyUILyr;
		tyLyrGen3 : tyUILyr;
		tyTxtWidthOffset : tyUITxt;
		tyNumWidthOffset : tyUINum;
		tyNumMagAutoDetSenTm : tyUINum;
		tyBtnAGVComEn : tyUIBtn;
		tyNumAutoLogoutTm : tyUINum;
		tyTxtLblAutoLogoutTm : tyUITxt;
		tyBtnAutoLogoutEn : tyUIBtn;
		tyBtnScannerEn : tyUIBtn;
		tyBtnLFBuzMute : tyUIBtn;
		tyDrpDnAGVComProtocol : tyUIDrpDn;
		tyDrpDnMagExchangeMode : tyUIDrpDn;
		tyBtnAGVSizeDisabled : tyUIBtn;
		tyNumAWPusherAtHm : tyUINum;
		tyNumTravFixtoFixPosOutlet : tyUINum;
		tyBtnDisableFMWarning : tyUIBtn;
		tyNumLMCFbTm : tyUINum;
		tyBtnMagWidthChkDis : tyUIBtn;
		tyNumMag1WidthChkDetDist : tyUINum;
		tyNumMag2WidthChkDetDist : tyUINum;
		tyNumMag3WidthChkDetDist : tyUINum;
		tyBtnDBAOnRgtSen : tyUIBtn;
		tyBtnHermesSvyEn : tyUIBtn;
		tyBtnRFIDEn : tyUIBtn;
		tyNumRFIDWrTO : tyUINum;
		tyNumTravLaneBOffset : tyUINum;
	END_STRUCT;
	tyLyrP1021McSetNetwork : 	STRUCT
		tyStringIPAddr : tyUIString;
		tyStringSubnetMask : tyUIString;
		tyBtnSave : tyUIBtn;
		tyBtnCancel : tyUIBtn;
		tyLyr : tyUILyr;
	END_STRUCT;
END_TYPE

(**)

TYPE
	tyLyrP1022McSetVCommSel : 	STRUCT
		tyBtnLF : tyUIBtn;
		tyBtnLCSLF : tyUIBtn;
		tyBtnLCSReqRcp : tyUIBtn;
		tyBtnLCSManageRcp : tyUIBtn;
		tyBtnLCSLiveDat : tyUIBtn;
		tyLyr : tyUILyr;
	END_STRUCT;
	tyLyrP1022McSetVCommLF : 	STRUCT
		tyBtnLeaderMc : tyUIBtn;
		tyBtnSectionLdr : tyUIBtn;
		tyBtnDBAOnWOAlign : tyUIBtn;
		tyBtnDSWidthChkEn : tyUIBtn;
		tyLyr : tyUILyr;
	END_STRUCT;
	tyLyrP1022McSetVCommSvy : 	STRUCT
		tyNumSndAliveTm : tyUINum;
		tyNumSvySystemPort : tyUINum;
		tyBtnConfiguration : tyUIBtn;
		tyBtnCheckAliveResponse : tyUIBtn;
		tyBtnBoardTracking : tyUIBtn;
		tyBtnQueryWorkOrderInfo : tyUIBtn;
		tyBtnSendWorkOrderInfo : tyUIBtn;
		tyBitmapMask : tyUIBitmap;
		tyLyr : tyUILyr;
	END_STRUCT;
END_TYPE

(**)

TYPE
	tyLyrP1023McSetHCommSel : 	STRUCT
		tyBtnSMEMA : tyUIBtn;
		tyBtnHermes : tyUIBtn;
		tyTxtHeader : tyUITxt;
		tyLyr : tyUILyr;
	END_STRUCT;
	tyLyrP1023McSetHCommSMEMA : 	STRUCT
		tyBtnGdSig : tyUIBtn;
		tyDrpDnSMEMAMod : tyUIDrpDn;
		tyLyr : tyUILyr;
	END_STRUCT;
	tyLyrP1023McSetHCommDSHermes : 	STRUCT
		tyNumLaneID : tyUINum;
		tyNumSvrPort : tyUINum;
		tyNumSndAliveTm : tyUINum;
		tyBtnCheckAliveResponse : tyUIBtn;
		tyBtnBoardForecast : tyUIBtn;
		tyBtnSendBoardInfo : tyUIBtn;
		tyBitmapMask : tyUIBitmap;
		tyLyr : tyUILyr;
	END_STRUCT;
END_TYPE

(**)

TYPE
	tyLyrP1024McSetAntiGap : 	STRUCT
		tyNumLftSenOff : tyUINum;
		tyNumRgtSenOff : tyUINum;
		tyNumMagConvEntOn : tyUINum;
		tyNumMagConvEntOff : tyUINum;
		tyNumMagConvPresentOn : tyUINum;
		tyNumMagConvPresentOff : tyUINum;
		tyLyr : tyUILyr;
	END_STRUCT;
END_TYPE

(**)

TYPE
	tyLyrP1025McSetAIVComm : 	STRUCT
		tyNumSvrPort : tyUINum;
		tyStringAllwClntIP : tyUIString;
		tyNumAllwClntPort : tyUINum;
		tyLyr : tyUILyr;
	END_STRUCT;
END_TYPE

(**)

TYPE
	tyLyrP1026McSetTeach : 	STRUCT
		tyBtn1 : tyUIBtn;
		tyBtn2 : tyUIBtn;
		tyBtn3 : tyUIBtn;
		tyBtn4 : tyUIBtn;
		tyLyr : tyUILyr;
	END_STRUCT;
	tyLyrP1026InOutletShutterFB : 	STRUCT
		tyStringStat : tyUILString;
		tyBtnOpen : tyUIBtn;
		tyBtnClose : tyUIBtn;
		tyLyr : tyUILyr;
	END_STRUCT;
END_TYPE

(**)

TYPE
	tyLyrP1027McSetUSBSetting : 	STRUCT
		tyVID : tyUINum;
		tyPID : tyUINum;
		tyBtnReset : tyUIBtn := (uiMaskRtStat:=0);
		tyBitError : tyUIBitmap;
		tyLyr : tyUILyr;
	END_STRUCT;
END_TYPE

(**)

TYPE
	tyLyrP1028McSetRS232Setting : 	STRUCT
		tyNumStartCode1 : tyUINum;
		tyNumStartCode2 : tyUINum;
		tyNumEndCode1 : tyUINum;
		tyNumEndCode2 : tyUINum;
		tyLyr : tyUILyr;
	END_STRUCT;
END_TYPE

(**)

TYPE
	tyLyrP1030MagSet : 	STRUCT
		tyStringRecipeNm : tyUIString;
		tyNumSltToSltDist : tyUINum;
		tyNumMaxSlt : tyUINum;
		tyBtnLifterMag1Slt1Pos : tyUIBtn;
		tyBtnLifterMag2Slt1Pos : tyUIBtn;
		tyBtnLifterMag3Slt1Pos : tyUIBtn;
		tyBtnLifterMag4Slt1Pos : tyUIBtn;
		tyBtnTravPosMag1 : tyUIBtn;
		tyBtnTravPosMag2 : tyUIBtn;
		tyBtnTravPosMag3 : tyUIBtn;
		tyBtnTravPosMag4 : tyUIBtn;
		tyBtnSave : tyUIBtn;
		tyBtnDelete : tyUIBtn;
		tyNumLifterMag1Slt1Pos : tyUINum;
		tyNumLifterMag2Slt1Pos : tyUINum;
		tyNumLifterMag3Slt1Pos : tyUINum;
		tyNumLifterMag4Slt1Pos : tyUINum;
		tyNumTravPosMag1 : tyUINum;
		tyNumTravPosMag2 : tyUINum;
		tyNumTravPosMag3 : tyUINum;
		tyNumTravPosMag4 : tyUINum;
		tyTxtLifMag3Slt1PosLbl : tyUITxt;
		tyTxtTravPosMag3Lbl : tyUITxt;
		tyTxtLifMag4Slt1PosLbl : tyUITxt;
		tyTxtTravPosMag4Lbl : tyUITxt;
		tyTableRecipe : tyUITable;
		tyDrpDnMagModel : tyUIDrpDn;
		tyTxtMagModel : tyUITxt;
		tyNumMagMaxBrdWidth : tyUINum;
		tyBtnSort : tyUIBtn;
		tyBtnSafetyBarDisabled : tyUIBtn;
		tyBtnMagHeightChkEn : tyUIBtn;
		tyBitmapBrder : tyUIBitmap;
	END_STRUCT;
END_TYPE

(**)

TYPE
	tyLyrP1031MagSetTeach : 	STRUCT
		tyBtn1 : tyUIBtn;
		tyBtn2 : tyUIBtn;
		tyBtn3 : tyUIBtn;
		tyBtn4 : tyUIBtn;
		tyLyr : tyUILyr;
		tyNumNewSlt : tyUINum;
	END_STRUCT;
	tyLyrP1031InOutletShutterFB : 	STRUCT
		tyStringStat : tyUILString;
		tyBtnOpen : tyUIBtn;
		tyBtnClose : tyUIBtn;
		tyLyr : tyUILyr;
	END_STRUCT;
END_TYPE

(**)

TYPE
	tyLyrP1040ProdSet : 	STRUCT
		tyHotspotShowLRcp : tyUIHotspot;
		tyStringRecipeNm : tyUILString;
		tyNumProdWidth2 : tyUINum;
		tyNumProdWidth : tyUINum;
		tyNumFirstSlt : tyUINum;
		tyNumLastSlt : tyUINum;
		tyNumPitch : tyUINum;
		tyDrpDnMcMode : tyUIDrpDn;
		tyDrpDnFlippedBrd : tyUIDrpDn;
		tyBtnToptoBtm : tyUIBtn;
		tyBtnLongBrd : tyUIBtn;
		tyBtnToXML : tyUIBtn;
		tyBtnFromXML : tyUIBtn;
		tyBtnSave : tyUIBtn;
		tyBtnDelete : tyUIBtn;
		tyStringSearch : tyUILString;
		tyTableRecipe : tyUITable;
		tyBtnSort : tyUIBtn;
		tyNumProdWidthRear : tyUINum;
		tyNumFirstSltRear : tyUINum;
		tyNumLastSltRear : tyUINum;
		tyNumPitchRear : tyUINum;
		tyNotQuadrupleLyr : tyUILyr;
		tyQuadrupleLyr : tyUILyr;
		tyNumMtrPshrExtSpd : tyUINum;
		tyNumMtrPshrExtTorq : tyUINum;
		tyNumPshrOffset : tyUINum;
		tyTxtPshrOffset : tyUITxt;
	END_STRUCT;
END_TYPE

(**)

TYPE
	tyLyrP1050LFSetLdr : 	STRUCT
		tyTable1List : tyUITable1;
		tyBtnEdit : tyUIBtn;
		tyBtnDelete : tyUIBtn;
		tyBtnOnline : tyUIBtn;
		tyBtnOffline : tyUIBtn;
		tyBtnShftUp : tyUIBtn;
		tyBtnShftDwn : tyUIBtn;
		tyNumBeforeOven : tyUINum;
		tyNumAfterOven : tyUINum;
		tyNumBeforeOven2 : tyUINum;
		tyNumAfterOven2 : tyUINum;
		tyLyr : tyUILyr;
	END_STRUCT;
	tyLyrP1050LFSetLdrEdit : 	STRUCT
		tyNumMcNum : tyUINum;
		tyStringIPAddr : tyUIString;
		tyBtnOk : tyUIBtn;
		tyBtnCancel : tyUIBtn;
		tyTxtLblInfoThirdParty : tyUITxt;
		tyLyr : tyUILyr;
	END_STRUCT;
END_TYPE

(**)

TYPE
	tyLyrP1080UsrMgmt : 	STRUCT
		tyDrpDnLvl : tyUIDrpDn;
		tyTableList : tyUITable1;
		tyBtnNewUsr : tyUIBtn;
		tyBtnEditDetail : tyUIBtn;
		tyBtnDeleteUsr : tyUIBtn;
		tyLyr : tyUILyr;
		tyBtnEditAccess : tyUIBtn;
	END_STRUCT;
	tyLyrP1080UsrMgmtAct : 	STRUCT
		tyStringUsrNm : tyUIString;
		tyStringPw : tyUIString;
		tyDrpDnLvl : tyUIDrpDn;
		tyBtnOk : tyUIBtn;
		tyBtnCancel : tyUIBtn;
		tyLyr : tyUILyr;
	END_STRUCT;
END_TYPE

(**)

TYPE
	tyLyrP1081UsrMgmtUsrAccessRgt : 	STRUCT
		tyBtnOps : tyUIBtn;
		tyBtnProdSel : tyUIBtn;
		tyBtnMagSel : tyUIBtn;
		tyBtnMcInfo : tyUIBtn;
		tyBtnAlm : tyUIBtn;
		tyBtnBffrInfo : tyUIBtn;
		tyBtnOvenInfo : tyUIBtn;
		tyBtnMagInfo : tyUIBtn;
		tyBtnLFCtrl : tyUIBtn;
		tyBtnManual : tyUIBtn;
		tyBtnSimu : tyUIBtn;
		tyBtnChgParam : tyUIBtn;
		tyBtnLFSet : tyUIBtn;
		tyBtnBackup : tyUIBtn;
		tyBtnLang : tyUIBtn;
		tyBtnMcSet : tyUIBtn;
		tyBtnProdSet : tyUIBtn;
		tyBtnMagSet : tyUIBtn;
		tyBtnManualFBOnly : tyUIBtn;
		tyStringNm : tyUIString;
		tyTxtTitle : tyUITxt;
		tyLyr : tyUILyr;
	END_STRUCT;
	tyLyrP1081UsrMgmtUsrAccessRgtSel : 	STRUCT
		tyDrpDnLevel : tyUIDrpDn;
		tyLyr : tyUILyr;
	END_STRUCT;
END_TYPE

(**)
(*Visu Property*)

TYPE
	tyVisu : 	STRUCT
		uiChgPage : UINT;
		uiCurrPage : UINT;
		uiSSaverTm : UINT;
		uiScreenSaverRemainTm : UINT;
		usiChgLang : USINT;
		usiCurrLang : USINT;
	END_STRUCT;
	tyKeypad : 	STRUCT
		tyStringTitle : tyUIString;
	END_STRUCT;
	tyTxtSnippets : 	STRUCT
		sLibraryNm : STRING[10];
		sUsrMgmtUsrLv1Nm : STRING[80];
		sUsrMgmtUsrLv2Nm : STRING[80];
		sUsrMgmtUsrLv3Nm : STRING[80];
	END_STRUCT;
END_TYPE
```

#### Visu_Layer.var
```iecst
(*Reference Common Layer*)
VAR
	p_tyC0001MotionStd : REFERENCE TO tyLyrC0001MotionStd; (*Motion Standard*)
END_VAR
(**)
VAR
	p_tyC0002FullMask : REFERENCE TO tyLyrC0002FullMask; (*Full Mask*)
END_VAR
(**)
VAR
	p_tyC0003DualMask : REFERENCE TO tyLyrC0003DualMask; (*Dual Mask*)
END_VAR
(**)
VAR
	p_tyC0004Navi : REFERENCE TO tyLyrC0004Navi; (*Navigation*)
END_VAR
(**)
VAR
	p_tyC0005Main : REFERENCE TO tyLyrC0005Main; (*Main*)
END_VAR
(**)
VAR
	p_tyC0006Set : REFERENCE TO tyLyrC0006Set; (*Setting*)
END_VAR
(**)
VAR
	p_tyC0007Notif : REFERENCE TO tyLyrC0007Notif; (*Notification*)
END_VAR
(**)
VAR
	p_tyC0008MsgBox : REFERENCE TO tyLyrC0008MsgBox; (*Message Box*)
END_VAR
(**)
VAR
	p_tyC0009Info : REFERENCE TO tyLyrC0009Info; (*Info*)
END_VAR
(**)
VAR
	p_tyC0010RcyMsg : REFERENCE TO tyLyrC0010RcyMsg; (*Recover Msg*)
END_VAR
(**)
VAR
	p_tyC0011RcpPopUp : REFERENCE TO tyLyrC0011RcpPopUp; (*254 Char Rcp Pop Up Layer*)
END_VAR
(**)
(*Reference Layer*)
VAR
	p_tyP0000SSaver : REFERENCE TO tyLyrP0000SSaver; (*Screen Saver*)
END_VAR
(**)
VAR
	p_tyP0001Startup : REFERENCE TO tyLyrP0001Startup; (*Startup*)
	p_tyP0001Initial : REFERENCE TO tyLyrP0001Initial; (*Startup*)
END_VAR
(**)
VAR
	p_tyP0002Menu : REFERENCE TO tyLyrP0002Menu; (*Menu*)
END_VAR
(**)
VAR
	p_tyP0100Login : REFERENCE TO tyLyrP0100Login; (*Login*)
	p_tyP0100Logout : REFERENCE TO tyLyrP0100Logout;
END_VAR
(**)
VAR
	p_tyP0200OpsGen : REFERENCE TO tyLyrP0200OpsGen; (*Operation*)
	p_tyP0200OpsDSCommB : REFERENCE TO tyLyrP0200OpsDSCommB;
	p_tyP0200OpsDSAVSMEMA : REFERENCE TO tyLyrP0200OpsDSAVSMEMA;
	p_tyP0200OpsDSBVSMEMA : REFERENCE TO tyLyrP0200OpsDSBVSMEMA;
	p_tyP0200OpsDSAVSMEMA1 : REFERENCE TO tyLyrP0200OpsDSAVSMEMA;
	p_tyP0200OpsDSBVSMEMA1 : REFERENCE TO tyLyrP0200OpsDSBVSMEMA;
	p_tyP0200OpsBypsInitConv : REFERENCE TO tyLyrP0200OpsBypsInitConv; (*Operation*)
	p_tyP0200OpsBarCodeScan : REFERENCE TO tyLyrP0200OpsBarCodeScan;
END_VAR
(**)
VAR
	p_tyP0201OpsTravLif : REFERENCE TO tyLyrP0201OpsTravLif;
	p_tyP0201TravLifIOMonitor : REFERENCE TO tyLyrP0201OpsTravLifIOMonitor;
	p_tyP0201TravLifBypsInitConv : REFERENCE TO tyLyrP0201OpsTravLifBypsInitConv;
	p_tyP0201Param : REFERENCE TO tyLyrP0201OpsParam;
	p_tyP0201OpsBarcodeScanner : REFERENCE TO tyLyrP0201OpsBarcodeScanner;
	p_tyP0201OpsCurrWorkOrder : REFERENCE TO tyLyrP0201OpsCurrWorkOrder;
	p_tyP0201OpsQueryBoardInfo : REFERENCE TO tyLyrP0201OpsQueryBoardInfo;
	p_tyP0201OpsQueryWorkOrder : REFERENCE TO tyLyrP0201OpsQueryWorkOrder;
END_VAR
(**)
VAR
	p_tyP0202Ops : REFERENCE TO tyLyrP0202Ops;
	p_tyP0202IOMonitor : REFERENCE TO tyLyrP0202IOMonitor;
	p_tyP0202BypsInitConv : REFERENCE TO tyLyrP0202BypsInitConv;
	p_tyP0202Param : REFERENCE TO tyLyrP0202OpsParam;
END_VAR
(**)
VAR
	p_tyP0203Ops : REFERENCE TO tyLyrP0203Ops;
	p_tyP0203IOMonitor : REFERENCE TO tyLyrP0203IOMonitor;
	p_tyP0203BypsInitConv : REFERENCE TO tyLyrP0203BypsInitConv;
	p_tyP0203Param : REFERENCE TO tyLyrP0203OpsParam;
END_VAR
(**)
VAR
	p_tyP0204Ops : REFERENCE TO tyLyrP0204Ops;
	p_tyP0204IOMonitor : REFERENCE TO tyLyrP0204IOMonitor;
	p_tyP0204BypsInitConv : REFERENCE TO tyLyrP0204BypsInitConv;
	p_tyP0204Param : REFERENCE TO tyLyrP0204OpsParam;
END_VAR
(**)
VAR
	p_tyP0205IOMonitor : REFERENCE TO tyLyrP0205IOMonitor; (*AIV IO MONITOR*)
END_VAR
(**)
VAR
	p_tyP0206Ops : REFERENCE TO tyLyrP0206Ops;
	p_tyP0206IOMonitor : REFERENCE TO tyLyrP0206IOMonitor;
	p_tyP0206BypsInitConv : REFERENCE TO tyLyrP0206BypsInitConv;
	p_tyP0206Param : REFERENCE TO tyLyrP0206OpsParam;
END_VAR
(**)
VAR
	p_tyP0300McInfo : REFERENCE TO tyLyrP0300McInfo; (*Operation*)
END_VAR
(**)
VAR
	p_tyP0400ProdSel : REFERENCE TO tyLyrP0400ProdSel; (*Product Selection*)
	p_tyP0400RcpDet : REFERENCE TO tyLyrP0400RcpDet; (*Product Selection_Recipe Detail*)
END_VAR
(**)
VAR
	p_tyP0410MagSel : REFERENCE TO tyLyrP0410MagSel; (*Magazine Selection*)
	p_tyP0410MagDet : REFERENCE TO tyLyrP0410MagDet;
END_VAR
(**)
VAR
	p_tyP0600Alm : REFERENCE TO tyLyrP0600Alm; (*Alarm*)
END_VAR
(**)
VAR
	p_tyP0700LFCtrl : REFERENCE TO tyLyrP0700LFCtrl; (*Master Slave*)
END_VAR
(**)
VAR
	p_tyP0800MagInfo1 : REFERENCE TO tyLyrP0800MagInfo1; (*Magazine Info*)
	p_tyP0800MagInfo2 : REFERENCE TO tyLyrP0800MagInfo2;
	p_tyP0800MagInfo3 : REFERENCE TO tyLyrP0800MagInfo3;
	p_tyP0800MagInfo4 : REFERENCE TO tyLyrP0800MagInfo3;
END_VAR
(**)
VAR
	p_tyP0900GenIn1 : REFERENCE TO tyLyrP0900GenIn1; (*General Input*)
	p_tyP0900GenIn2 : REFERENCE TO tyLyrP0900GenIn2;
END_VAR
(**)
VAR
	p_tyP0910GenOut : REFERENCE TO tyLyrP0910GenOut; (*General Output*)
	p_tyP0910GenOutCurtainSen : REFERENCE TO tyLyrP0910GenOutCurtainSen; (*General Output*)
END_VAR
(**)
VAR
	p_tyP0920MtrNPneuCtrl : REFERENCE TO tyLyrP0920MtrNPneuCtrl; (*Motor And Pneumatic Control*)
	p_tyP0920MtrNPneuCtrlPneu : REFERENCE TO tyLyrP0920MtrNPneuCtrlPneu;
END_VAR
(**)
VAR
	p_tyP0921InletShutterCom : REFERENCE TO tyLyrP0921InletShutterCom;
	p_tyP0921InletShutterDC : REFERENCE TO tyLyrP0921InletShutterDC;
	p_tyP0921InletShutterFB : REFERENCE TO tyLyrP0921InletShutterFB;
	p_tyP0921OutletShutterCom : REFERENCE TO tyLyrP0921OutletShutterCom;
	p_tyP0921OutletShutterDC : REFERENCE TO tyLyrP0921OutletShutterDC;
	p_tyP0921OutletShutterFB : REFERENCE TO tyLyrP0921OutletShutterFB;
	p_tyP0921OutletShutterDis : REFERENCE TO tyLyrP0921OutletShutterDis;
END_VAR
(**)
VAR
	p_tyP0923LftSafetyBarCom : REFERENCE TO tyLyrP0923LftSafetyBarCom;
	p_tyP0923LftSafetyBarDC : REFERENCE TO tyLyrP0923LftSafetyBarDC;
	p_tyP0923LftSafetyBarFB : REFERENCE TO tyLyrP0923LftSafetyBarFB;
	p_tyP0923RgtSafetyBarCom : REFERENCE TO tyLyrP0923RgtSafetyBarCom;
	p_tyP0923RgtSafetyBarDC : REFERENCE TO tyLyrP0923RgtSafetyBarDC;
	p_tyP0923RgtSafetyBarFB : REFERENCE TO tyLyrP0923RgtSafetyBarFB;
END_VAR
(**)
VAR
	p_tyP0924TrolleyLckCom : REFERENCE TO tyLyrP0924TrolleyLckCom;
	p_tyP0924TrolleyLckDC : REFERENCE TO tyLyrP0924TrolleyLckDC;
	p_tyP0924TrolleyLckFB : REFERENCE TO tyLyrP0924TrolleyLckFB;
END_VAR
(**)
VAR
	p_tyP0930Mag1ConvCom : REFERENCE TO tyLyrP0930Mag1ConvCom;
	p_tyP0930Mag1ConvDC : REFERENCE TO tyLyrP0930Mag1ConvDC;
	p_tyP0930Mag1ConvFB : REFERENCE TO tyLyrP0930Mag1ConvFB;
END_VAR
(**)
VAR
	p_tyP0931Mag2ConvCom : REFERENCE TO tyLyrP0931Mag2ConvCom;
	p_tyP0931Mag2ConvDC : REFERENCE TO tyLyrP0931Mag2ConvDC;
	p_tyP0931Mag2ConvFB : REFERENCE TO tyLyrP0931Mag2ConvFB;
END_VAR
(**)
VAR
	p_tyP0932Mag3ConvCom : REFERENCE TO tyLyrP0932Mag3ConvCom;
	p_tyP0932Mag3ConvDC : REFERENCE TO tyLyrP0932Mag3ConvDC;
	p_tyP0932Mag3ConvFB : REFERENCE TO tyLyrP0932Mag3ConvFB;
END_VAR
(**)
VAR
	p_tyP0933PullConvCom : REFERENCE TO tyLyrP0933PullConvCom;
	p_tyP0933PullConvDC : REFERENCE TO tyLyrP0933PullConvDC;
	p_tyP0933PullConvFB : REFERENCE TO tyLyrP0933PullConvFB;
END_VAR
(**)
VAR
	p_tyP0934AW : REFERENCE TO tyLyrP0934AW;
END_VAR
(**)
VAR
	p_tyP0935Lifter : REFERENCE TO tyLyrP0935Lifter; (*Lifter*)
END_VAR
(**)
VAR
	p_tyP0936Trav : REFERENCE TO tyLyrP0936Trav;
END_VAR
(**)
VAR
	p_tyP0937AWPushOrPuller : REFERENCE TO tyLyrP0937AWPushOrPuller;
	p_tyP0937InOutletShutterFB : REFERENCE TO tyLyrP0937InOutletShutterFB;
END_VAR
(**)
VAR
	p_tyP0939Mag4ConvCom : REFERENCE TO tyLyrP0939Mag4ConvCom;
	p_tyP0939Mag4ConvDC : REFERENCE TO tyLyrP0939Mag4ConvDC;
	p_tyP0939Mag4ConvFB : REFERENCE TO tyLyrP0939Mag4ConvFB;
END_VAR
(**)
VAR
	p_tyP0940CommCtrlDSSMEMAA : REFERENCE TO tyLyrP0940CommCtrlDSSMEMA; (*SMEMA Control*)
	p_tyP0940CommCtrlDSSMEMAB : REFERENCE TO tyLyrP0940CommCtrlDSSMEMA;
	p_tyP0940CommCtrlSOT : REFERENCE TO tyLyrP0940SOTComm;
END_VAR
(**)
VAR
	p_tyP0950Simu : REFERENCE TO tyLyrP0950Simu; (*Simulation*)
	p_tyP0950SimuAGVtoMC : REFERENCE TO tyLyrP0950SimuAGVToMC; (*SMEMA Control*)
	p_tyP0950SimuMCtoAGV : REFERENCE TO tyLyrP0950SimuMCToAGV; (*SMEMA Control*)
END_VAR
(**)
VAR
	p_tyP1000Lang : REFERENCE TO tyLyrP1000Lang; (*Language And Setup*)
END_VAR
(**)
VAR
	p_tyP1020McSetNavi : REFERENCE TO tyLyrP1020McSetNavi; (*Machine Setting*)
END_VAR
(**)
VAR
	p_tyP1021McSetGen : REFERENCE TO tyLyrP1021McSetGen;
	p_tyP1021McSetNetwork : REFERENCE TO tyLyrP1021McSetNetwork;
END_VAR
(**)
VAR
	p_tyP1022McSetVCommSel : REFERENCE TO tyLyrP1022McSetVCommSel; (*Machine Setting - US Commnunication SMEMA*)
	p_tyP1022McSetVCommLF : REFERENCE TO tyLyrP1022McSetVCommLF; (*Machine Setting - US Commnunication SMEMA*)
	p_tyP1022McSetVCommSvy : REFERENCE TO tyLyrP1022McSetVCommSvy; (*Machine Setting - US Commnunication SMEMA*)
END_VAR
(**)
VAR
	p_tyP1023McSetHCommDSSel : REFERENCE TO tyLyrP1023McSetHCommSel;
	p_tyP1023McSetHCommDSSMEMA : REFERENCE TO tyLyrP1023McSetHCommSMEMA;
	p_tyP1023McSetHCommDSHermes : REFERENCE TO tyLyrP1023McSetHCommDSHermes;
END_VAR
(**)
VAR
	p_tyP1024McSetAntiGap : REFERENCE TO tyLyrP1024McSetAntiGap;
END_VAR
(**)
VAR
	p_tyP1025McSetAIVComm : REFERENCE TO tyLyrP1025McSetAIVComm;
END_VAR
(**)
VAR
	p_tyP1026McSetTeach : REFERENCE TO tyLyrP1026McSetTeach;
	p_tyP1026InOutletShutterFB : REFERENCE TO tyLyrP1026InOutletShutterFB;
END_VAR
(**)
VAR
	p_tyP1027McSetUSBSetting : REFERENCE TO tyLyrP1027McSetUSBSetting;
END_VAR
(**)
VAR
	p_tyP1028McSetRS232Setting : REFERENCE TO tyLyrP1028McSetRS232Setting;
END_VAR
(**)
VAR
	p_tyP1030MagSet : REFERENCE TO tyLyrP1030MagSet; (*Magazine Setting*)
END_VAR
(**)
VAR
	p_tyP1031MagSetTeach : REFERENCE TO tyLyrP1031MagSetTeach;
	p_tyP1031InOutletShutterFB : REFERENCE TO tyLyrP1031InOutletShutterFB;
END_VAR
(**)
VAR
	p_tyP1040ProdSet : REFERENCE TO tyLyrP1040ProdSet; (*Product Setting*)
END_VAR
(**)
VAR
	p_tyP1050LFSetLdr : REFERENCE TO tyLyrP1050LFSetLdr;
	p_tyP1050LFSetLdrEdit : REFERENCE TO tyLyrP1050LFSetLdrEdit;
END_VAR
(**)
VAR
	p_tyP1080UsrMgmt : REFERENCE TO tyLyrP1080UsrMgmt; (*User Management*)
	p_tyP1080UsrMgmtAct : REFERENCE TO tyLyrP1080UsrMgmtAct;
END_VAR
(**)
VAR
	p_tyP1081UsrMgmtUsrAccessRgt : REFERENCE TO tyLyrP1081UsrMgmtUsrAccessRgt;
	p_tyP1081UsrMgmtUsrAccessRgtSel : REFERENCE TO tyLyrP1081UsrMgmtUsrAccessRgtSel;
END_VAR
(**)
(*Visu Property*)
VAR
	p_tyTxtSnippets : REFERENCE TO tyTxtSnippets; (*Text Snippets*)
	p_tyKeypad : REFERENCE TO tyKeypad; (*Keypad*)
	p_tyVisu : REFERENCE TO tyVisu; (*Visualization Properties*)
END_VAR
(**)
```

### Startup.typ
```iecst
(*2019-04-04*)
(**)

TYPE
	eStartupAction :
		(
		StartupActIdle,
		StartupActRun
		);
	eStartupStep :
		(
		StartupStepUsrFolder,
		StartupStepParameter,
		StartupStepGetHWInfo,
		StartupStepLibVer,
		StartupStepRecipe,
		StartupStepUsrMgmt,
		StartupStepBffr,
		StartupStepAlarm,
		StartupStepSerial,
		StartupStepHermes,
		StartupStepSDOWrite,
		StartupStepSetupUI,
		StartupStepAutoRcp,
		StartupStepDone
		);
END_TYPE
```

### Startup.var
```iecst
(*2020-09-16*)
(**)
(*Action & State & Status*)
VAR
	p_StartupStat : UDINT;
	p_StartupStatus : UDINT;
	p_StartupStatTxt : UDINT;
END_VAR
(**)
(*Alarm*)
(**)
(*Output*)
VAR
	p_StartupRun : UDINT;
	p_StartupUsrFolderAct : UDINT;
	p_StartupHWInfoAct : UDINT;
	p_StartupLibVerAct : UDINT;
	p_StartupNtParamAct : UDINT;
	p_StartupMcParamAct : UDINT;
	p_StartupProdRcpAct : UDINT;
	p_StartupMpProdRcpAct : UDINT;
	p_StartupMagRcpAct1 : UDINT;
	p_StartupMagRcpAct : UDINT;
	p_StartupUsrMgmtAct : UDINT;
	p_StartupBuffer1Act : UDINT;
	p_StartupBuffer2Act : UDINT;
	p_StartupBuffer3Act : UDINT;
	p_StartupBuffer4Act : UDINT;
	p_StartupAlarmAct : UDINT;
	p_StartupUIAct : UDINT;
	p_StartupAWPushPulAct : UDINT;
	p_StartupAWAct : UDINT;
	p_StartupTravAct : UDINT;
	p_StartupLifterAct : UDINT;
	p_StartupHermesAct : UDINT;
	p_StartupRmtHermesAct : UDINT;
	p_StartupDSHermesAAct : UDINT;
	p_StartupDSHermesBAct : UDINT;
	p_StartupStep : UDINT;
	p_StartupFrmAct : UDINT;
	p_StartupUSBAct : UDINT;
	p_StartupNtSettingsLoadDone : UDINT;
	p_StartupUISettingsLoadDone : UDINT;
	p_StartupSvyHermesAct : UDINT;
	p_StartupWaitDecision : UDINT;
	p_StartupAutoRcpsAct : UDINT;
	p_StartupStepTxt : UDINT;
	p_StartupGetConfigDone : UDINT;
	p_StartupMismatchSetConfigDone : UDINT;
	p_StartupServoPPAct : UDINT;
END_VAR
```

### Program Logical/Startup/Startup

#### InputRef.var
```iecst
(*2020-09-22*)
(**)
(*General*)
VAR
	p_eAct : REFERENCE TO eStartupAction;
	p_tyNtParamCurr : REFERENCE TO tyNtParam;
	p_tyMcParamCurr : REFERENCE TO tyMcParam;
	p_bUIMismatchOverWriteConfig : REFERENCE TO BOOL;
	p_bUITempAddrFillDone : REFERENCE TO BOOL;
	p_bUIChgConfigDone : REFERENCE TO BOOL;
	p_bUIOverwriteIP : REFERENCE TO BOOL;
	p_bUIOverwriteSubnet : REFERENCE TO BOOL;
	p_bUIOverwriteEthMode : REFERENCE TO BOOL;
	p_bUIReadWorkOrder : REFERENCE TO BOOL;
	p_bUISkipWorkOrder : REFERENCE TO BOOL;
END_VAR
```

#### InputRef_Link.var
```iecst
(*2020-09-22*)
(**)
(*User Folder*)
VAR
	p_eUsrFolderStat : REFERENCE TO eUsrFolderAction;
	p_eUsrFolderStatus : REFERENCE TO eFBStatus;
END_VAR
(**)
(*Hardware Info*)
VAR
	p_eHWInfoStat : REFERENCE TO eHWInfoAction;
	p_eHWInfoStatus : REFERENCE TO eFBStatus;
	p_sHWInfoIPAddr : REFERENCE TO STRING[15];
	p_sHWInfoSubnetMask : REFERENCE TO STRING[15];
	p_udiHWInfoEthMode : REFERENCE TO UDINT;
END_VAR
(**)
(*Library Version*)
VAR
	p_eLibVerStat : REFERENCE TO eLibVerAction;
	p_eLibVerStatus : REFERENCE TO eFBStatus;
END_VAR
(**)
(*Nutek Parameter*)
VAR
	p_eNtParamStat : REFERENCE TO eNtParamAction;
	p_eNtParamStatus : REFERENCE TO eFBStatus;
END_VAR
(**)
(*Machine Parameter*)
VAR
	p_eMcParamStat : REFERENCE TO eMcParamAction;
	p_eMcParamStatus : REFERENCE TO eFBStatus;
END_VAR
(**)
(*Product Recipe*)
VAR
	p_eProdRcpStat : REFERENCE TO eProdRcpAction;
	p_eProdRcpStatus : REFERENCE TO eFBStatus;
END_VAR
(**)
(*Mp Product Recipe*)
VAR
	p_eMpProdRcpStat : REFERENCE TO eMpProdRcpAction;
	p_eMpProdRcpStatus : REFERENCE TO eFBStatus;
END_VAR
(**)
(*Magazine Recipe*)
VAR
	p_eMagRcpStat : REFERENCE TO eMagRcpAction;
	p_eMagRcpStatus : REFERENCE TO eFBStatus;
	p_eMagRcpStat1 : REFERENCE TO eMagRcpAction;
	p_eMagRcpStatus1 : REFERENCE TO eFBStatus;
END_VAR
(**)
(*User Management*)
VAR
	p_eUsrMgmtStat : REFERENCE TO eUsrMgmtAction;
	p_eUsrMgmtStatus : REFERENCE TO eFBStatus;
END_VAR
(**)
(*Buffer*)
VAR
	p_eBuffer1Stat : REFERENCE TO eBufferAction;
	p_eBuffer1Status : REFERENCE TO eFBStatus;
	p_bMagPresentSensor1 : REFERENCE TO BOOL;
	p_bMagPresent1 : REFERENCE TO BOOL;
END_VAR
(**)
VAR
	p_eBuffer2Stat : REFERENCE TO eBufferAction;
	p_eBuffer2Status : REFERENCE TO eFBStatus;
	p_bMagPresentSensor2 : REFERENCE TO BOOL;
	p_bMagPresent2 : REFERENCE TO BOOL;
END_VAR
(**)
VAR
	p_eBuffer3Stat : REFERENCE TO eBufferAction;
	p_eBuffer3Status : REFERENCE TO eFBStatus;
	p_bMagPresentSensor3 : REFERENCE TO BOOL;
	p_bMagPresent3 : REFERENCE TO BOOL;
END_VAR
(**)
VAR
	p_eBuffer4Stat : REFERENCE TO eBufferAction;
	p_eBuffer4Status : REFERENCE TO eFBStatus;
	p_bMagPresentSensor4 : REFERENCE TO BOOL;
	p_bMagPresent4 : REFERENCE TO BOOL;
END_VAR
(**)
(*Alarm Log*)
VAR
	p_eAlarmStat : REFERENCE TO eAlarmAction;
	p_eAlarmStatus : REFERENCE TO eFBStatus;
END_VAR
(**)
(*Hermes*)
VAR
	p_eHermesStat : REFERENCE TO eHermesAction;
	p_eHermesStatus : REFERENCE TO eFBStatus;
	p_eRmtHermesStat : REFERENCE TO eHermesAction;
	p_eRmtHermesStatus : REFERENCE TO eFBStatus;
	p_eDSHermesAStat : REFERENCE TO eHermesAction;
	p_eDSHermesAStatus : REFERENCE TO eFBStatus;
	p_eDSHermesBStat : REFERENCE TO eHermesAction;
	p_eDSHermesBStatus : REFERENCE TO eFBStatus;
	p_eSvyHermesStat : REFERENCE TO eHermesAction;
	p_eSvyHermesStatus : REFERENCE TO eFBStatus;
END_VAR
(**)
(*Auto Width Pusher/Puller*)
VAR
	p_eAWPushOrPullerStat : REFERENCE TO eAWAction;
	p_eAWPushOrPullerStatus : REFERENCE TO eFBStatus;
END_VAR
(**)
(*Auto Width*)
VAR
	p_eAWStat : REFERENCE TO eAWAction;
	p_eAWStatus : REFERENCE TO eFBStatus;
END_VAR
(**)
(*Traverser*)
VAR
	p_eTravStat : REFERENCE TO eTravAction;
	p_eTravStatus : REFERENCE TO eFBStatus;
END_VAR
(**)
(*Lifter*)
VAR
	p_eLifterStat : REFERENCE TO eLifterAction;
	p_eLifterStatus : REFERENCE TO eFBStatus;
END_VAR
(**)
(*Servo Puller/Pusher*)
VAR
	p_eServoPPStat : REFERENCE TO ePullerPusherAction;
	p_eServoPPStatus : REFERENCE TO eFBStatus;
END_VAR
(**)
(*User Interface*)
VAR
	p_eUIStat : REFERENCE TO eUIAction;
	p_eUIStatus : REFERENCE TO eFBStatus;
END_VAR
(**)
(*Serial Log*)
VAR
	p_eFrmStat : REFERENCE TO eFrmAction;
	p_eFrmStatus : REFERENCE TO eFBStatus;
	p_eUSBStat : REFERENCE TO eUSBRdrAction;
	p_eUSBStatus : REFERENCE TO eFBStatus;
END_VAR
(* *)
VAR
	p_bNtParamAutoRcpPrep : REFERENCE TO BOOL;
	p_eAutoRcpStat : REFERENCE TO eAutoRcpAction;
	p_eAutoRcpStatus : REFERENCE TO eFBStatus;
END_VAR
```

#### Local.var
```iecst
(*2020-09-22*)
(**)
(*Local Action, State & Status*)
VAR
	eAct : eStartupAction := StartupActIdle;
	eStat : eStartupAction := StartupActIdle;
	eStatus : eFBStatus := Idle;
	sStatTxt : STRING[200] := '';
	a_sStatText : ARRAY[0..50] OF STRING[200] := ['Idling','Running Startup',49('')];
END_VAR
(**)
(*Local Alarm*)
(**)
(*Local Output*)
VAR
	bRun : BOOL;
	eUsrFolderAct : eUsrFolderAction;
	eHWInfoAct : eHWInfoAction;
	eLibVerAct : eLibVerAction;
	eNtParamAct : eNtParamAction;
	eMcParamAct : eMcParamAction;
	eProdRcpAct : eProdRcpAction;
	eMpProdRcpAct : eMpProdRcpAction;
	eMagRcpAct : eMagRcpAction;
	eMagRcpAct1 : eMagRcpAction;
	eUsrMgmtAct : eUsrMgmtAction;
	eBuffer1Act : eBufferAction;
	eBuffer2Act : eBufferAction;
	eBuffer3Act : eBufferAction;
	eBuffer4Act : eBufferAction;
	eAlarmAct : eAlarmAction;
	eUIAct : eUIAction;
	eAWPushPulAct : eAWAction;
	eAWAct : eAWAction;
	eTravAct : eTravAction;
	eServoPPAct : ePullerPusherAction;
	eLifterAct : eLifterAction;
	eFrmAct : eFrmAction;
	eUSBAct : eUSBRdrAction;
	eHermesAct : eHermesAction;
	eRmtHermesAct : eHermesAction;
	eSvyHermesAct : eHermesAction;
	eAutoRcpAct : eAutoRcpAction;
	eDSHermesAAct : eHermesAction;
	eDSHermesBAct : eHermesAction;
	eStartupStep1 : eStartupStep;
	bNtSettingsLoadDone : BOOL := FALSE;
	bUISettingsLoadDone : BOOL;
	sStepTxt : STRING[80];
	a_sStepText : ARRAY[0..11] OF STRING[80] := ['Creating User Folder','Reading Parameter','Getting Hardware Info','Checking Library Version','Reading Recipe List','Reading User Management List','Reading Buffer / Magazine Data','Setting Up Alarm','Setting Up Hermes','Writing Data To Servo Motor','Setting Up User Interface','Done'];
END_VAR
(**)
(*Local Input*)
VAR
	tyNtParamCurr : tyNtParam;
	tyMcParamCurr : tyMcParam;
	bMismatchOverWriteConfig : BOOL;
	bMismatchSetConfigDone : BOOL;
	bWaitDecision : BOOL;
	bTempAddrFillDone : BOOL;
	bChgConfigDone : BOOL;
	bOverwriteIP : BOOL;
	bOverwriteSubnet : BOOL;
	bOverwriteEthMode : BOOL;
	bGetConfigDone : BOOL;
END_VAR
(**)
(*Local*)
VAR
	bInitDone : BOOL;
	bInitialDone : BOOL;
	usiStep : USINT;
END_VAR
```

#### Act_InitGlobal.st
```iecst
(** 2020-09-22 **)
ACTION Act_InitGlobal:

	(* Always Change If Project Change *)

	//Pass Data To Link

	//Pass Data To Internal Use
	p_eAct ACCESS p_UIStartupAct;
	p_tyNtParamCurr ACCESS p_NtParamCurr;
	p_tyMcParamCurr ACCESS p_McParamCurr;

	p_bUIMismatchOverWriteConfig ACCESS p_UIMismatchOverWriteConfig;
	p_bUITempAddrFillDone ACCESS p_UITempAddrFillDone;
	p_bUIChgConfigDone ACCESS p_UIIPConfigChgDone;
	p_bUIOverwriteIP ACCESS p_UIOverwriteIP;
	p_bUIOverwriteSubnet ACCESS p_UIOverwriteSubnet;
	p_bUIOverwriteEthMode ACCESS p_UIOverwriteEthMode;

	p_eUsrFolderStat ACCESS p_UsrFolderStat;
	p_eUsrFolderStatus ACCESS p_UsrFolderStatus;

	p_eHWInfoStat ACCESS p_HWInfoStat;
	p_eHWInfoStatus ACCESS p_HWInfoStatus;
	p_sHWInfoIPAddr ACCESS p_HWInfoIPAddr;
	p_sHWInfoSubnetMask ACCESS p_HWInfoSubnetMask;
	p_udiHWInfoEthMode ACCESS p_HWInfoEthMode;

	p_eLibVerStat ACCESS p_LibVerStat;
	p_eLibVerStatus ACCESS p_LibVerStatus;

	p_eNtParamStat ACCESS p_NtParamStat;
	p_eNtParamStatus ACCESS p_NtParamStatus;

	p_eMcParamStat ACCESS p_McParamStat;
	p_eMcParamStatus ACCESS p_McParamStatus;

	p_eProdRcpStat ACCESS p_ProdRcpStat;
	p_eProdRcpStatus ACCESS p_ProdRcpStatus;

	p_eMpProdRcpStat ACCESS p_MpProdRcpStat;
	p_eMpProdRcpStatus ACCESS p_MpProdRcpStatus;

	p_eMagRcpStat ACCESS p_MagRcpStat;
	p_eMagRcpStatus ACCESS p_MagRcpStatus;
	p_eMagRcpStat1 ACCESS p_MagRcpStat1;
	p_eMagRcpStatus1 ACCESS p_MagRcpStatus1;

	p_eUsrMgmtStat ACCESS p_UsrMgmtStat;
	p_eUsrMgmtStatus ACCESS p_UsrMgmtStatus;

	p_eBuffer1Stat ACCESS p_Buffer1Stat;
	p_eBuffer1Status ACCESS p_Buffer1Status;
	p_bMagPresentSensor1 ACCESS p_DIMagPresentSen1;
	p_bMagPresent1 ACCESS p_Buffer1MagPresent;

	p_eBuffer2Stat ACCESS p_Buffer2Stat;
	p_eBuffer2Status ACCESS p_Buffer2Status;
	p_bMagPresentSensor2 ACCESS p_DIMagPresentSen2;
	p_bMagPresent2 ACCESS p_Buffer2MagPresent;

	p_eBuffer3Stat ACCESS p_Buffer3Stat;
	p_eBuffer3Status ACCESS p_Buffer3Status;
	p_bMagPresentSensor3 ACCESS p_DIMagPresentSen3;
	p_bMagPresent3 ACCESS p_Buffer3MagPresent;

	p_eBuffer4Stat ACCESS p_Buffer4Stat;
	p_eBuffer4Status ACCESS p_Buffer4Status;
	p_bMagPresentSensor4 ACCESS p_DIMagPresentSen4;
	p_bMagPresent4 ACCESS p_Buffer4MagPresent;

	p_eAlarmStat ACCESS p_AlarmStat;
	p_eAlarmStatus ACCESS p_AlarmStatus;

	p_eHermesStat ACCESS p_HermesStat;
	p_eHermesStatus ACCESS p_HermesStatus;

	p_eRmtHermesStat ACCESS p_RmtHermesStat;
	p_eRmtHermesStatus ACCESS p_RmtHermesStatus;

	p_eDSHermesAStat ACCESS p_DSHermesAStat;
	p_eDSHermesAStatus ACCESS p_DSHermesAStatus;

	p_eDSHermesBStat ACCESS p_DSHermesBStat;
	p_eDSHermesBStatus ACCESS p_DSHermesBStatus;
	p_eSvyHermesStat ACCESS p_SvyHermesStat;//new for Hermes 1.3
	p_eSvyHermesStatus ACCESS p_SvyHermesStatus;//new for Hermes 1.3
	p_bUISkipWorkOrder ACCESS p_UISkipWorkOrder;//new for Hermes 1.3
	p_bUIReadWorkOrder ACCESS p_UIReadWorkOrder;//new for Hermes 1.3

	p_eAWPushOrPullerStat ACCESS p_AWPushOrPullerStat;
	p_eAWPushOrPullerStatus ACCESS p_AWPushOrPullerStatus;

	p_eAWStat ACCESS p_AWOpenStat;
	p_eAWStatus ACCESS p_AWOpenStatus;

	p_eTravStat ACCESS p_TravStat;
	p_eTravStatus ACCESS p_TravStatus;

	p_eLifterStat ACCESS p_LifterBtmStat;
	p_eLifterStatus ACCESS p_LifterBtmStatus;

	p_eUIStat ACCESS p_UIStat;
	p_eUIStatus ACCESS p_UIStatus;

	p_eUSBStat ACCESS p_USBRdrStat;
	p_eUSBStatus ACCESS p_USBRdrStatus;

	p_eFrmStat ACCESS p_FrmStat;
	p_eFrmStatus ACCESS p_FrmStatus;

	p_eServoPPStat ACCESS p_PPStat;
	p_eServoPPStatus ACCESS p_PPStatus;

	p_bNtParamAutoRcpPrep ACCESS p_NtParamAutoRcpPrep;
	p_eAutoRcpStat ACCESS p_AutoRcpStat;
	p_eAutoRcpStatus ACCESS p_AutoRcpStatus;

	(* Always Change If Project Change *)

END_ACTION
```

#### Act_Main.st
```iecst
(** 2019-03-28 **)
ACTION Act_Main:

	//Main
	CASE eStat OF

		StartupActIdle:
			IF eStatus <> Idle THEN	//Reset Data
				//Private
				eStartupStep1	:= StartupStepUsrFolder;
				bRun			:= FALSE;
				usiStep			:= 0;

				sStatTxt	:= a_sStatText[eStat];

			END_IF

			eStatus	:= Idle;

		StartupActRun:
			IF eStatus = Idle OR eStatus = Busy THEN

				eStatus	:= Busy;

				sStatTxt	:= a_sStatText[eStat];

				bRun	:= TRUE;

				CASE eStartupStep1 OF

					StartupStepUsrFolder:
						Act_Main_UsrFolder;

					StartupStepParameter:
						Act_Main_Parameter;

					StartupStepGetHWInfo:
						Act_Main_GetHWInfo;

					StartupStepLibVer:
						Act_Main_LibVer;

					StartupStepRecipe:
						Act_Main_Recipe;

					StartupStepAutoRcp:
						IF p_bNtParamAutoRcpPrep THEN
							Act_Main_AutoRcp;
						ELSE
							eStartupStep1:= StartupStepUsrMgmt;
						END_IF
					StartupStepUsrMgmt:
						Act_Main_UsrMgmt;

					StartupStepBffr:
						Act_Main_Bffr;

					StartupStepAlarm:
						Act_Main_Alarm;

					StartupStepSerial:
						Act_Main_Serial;

					StartupStepHermes:
						Act_Main_Hermes;

					StartupStepSDOWrite:
						IF DiagCpuIsSimulated() = FALSE THEN
							Act_Main_SDOWrite;
						ELSE
							eStartupStep1	:= StartupStepSetupUI;
						END_IF

					StartupStepSetupUI:
						Act_Main_SetupUI;

					StartupStepDone:
						Act_Main_Done;

				END_CASE

				sStepTxt	:= a_sStepText[eStartupStep1];

			END_IF

	END_CASE

END_ACTION
```

#### Init.st
```iecst
(** 2019-05-04 **)
PROGRAM _INIT

	(* Always Change If Project Change *)

	//Pass Address To External Use
	p_StartupStat		:= ADR(eStat);
	p_StartupStatus		:= ADR(eStatus);
	p_StartupStatTxt	:= ADR(sStatTxt);

	//Alarm

	//Output
	p_StartupRun				:= ADR(bRun);
	p_StartupUsrFolderAct		:= ADR(eUsrFolderAct);
	p_StartupHWInfoAct			:= ADR(eHWInfoAct);
	p_StartupLibVerAct			:= ADR(eLibVerAct);
	p_StartupNtParamAct			:= ADR(eNtParamAct);
	p_StartupMcParamAct			:= ADR(eMcParamAct);
	p_StartupProdRcpAct			:= ADR(eProdRcpAct);
	p_StartupMpProdRcpAct		:= ADR(eMpProdRcpAct);
	p_StartupMagRcpAct			:= ADR(eMagRcpAct);
	p_StartupMagRcpAct1			:= ADR(eMagRcpAct1);
	p_StartupUsrMgmtAct			:= ADR(eUsrMgmtAct);
	p_StartupBuffer1Act			:= ADR(eBuffer1Act);
	p_StartupBuffer2Act			:= ADR(eBuffer2Act);
	p_StartupBuffer3Act			:= ADR(eBuffer3Act);
	p_StartupBuffer4Act			:= ADR(eBuffer4Act);
	p_StartupAlarmAct			:= ADR(eAlarmAct);
	p_StartupUIAct				:= ADR(eUIAct);
	p_StartupAWAct				:= ADR(eAWAct);
	p_StartupAWPushPulAct		:= ADR(eAWPushPulAct);
	p_StartupTravAct			:= ADR(eTravAct);
	p_StartupLifterAct			:= ADR(eLifterAct);
	p_StartupHermesAct			:= ADR(eHermesAct);
	p_StartupRmtHermesAct		:= ADR(eRmtHermesAct);
	p_StartupDSHermesAAct		:= ADR(eDSHermesAAct);
	p_StartupDSHermesBAct		:= ADR(eDSHermesBAct);
	p_StartupStep				:= ADR(eStartupStep1);
	p_StartupUSBAct				:= ADR(eUSBAct);
	p_StartupFrmAct				:= ADR(eFrmAct);
	p_StartupServoPPAct			:= ADR(eServoPPAct);

	p_StartupNtSettingsLoadDone	:= ADR(bNtSettingsLoadDone);
	p_StartupUISettingsLoadDone := ADR(bUISettingsLoadDone);
	p_StartupStepTxt			:= ADR(sStepTxt);
	p_StartupSvyHermesAct		:= ADR(eSvyHermesAct); //new for Hermes 1.3
	p_StartupWaitDecision    	:= ADR(bWaitDecision); //new for Hermes 1.3
	p_StartupAutoRcpsAct		:= ADR(eAutoRcpAct);

	p_StartupGetConfigDone			:= ADR(bGetConfigDone);
	p_StartupMismatchSetConfigDone	:= ADR(bMismatchSetConfigDone);
	(* Always Change If Project Change *)

END_PROGRAM
```

#### Act_Main_AutoRcp.st
```iecst
(** 2019-05-04 **)
ACTION Act_Main_AutoRcp:

	CASE usiStep OF
		0:
			eAutoRcpAct	:= AutoRcpActCreateDir;

			IF (p_eAutoRcpStatus = Done) AND (p_eAutoRcpStat = AutoRcpActCreateDir) THEN

				eAutoRcpAct		:= AutoRcpActIdle;
				usiStep			:= 1;

			ELSIF p_eAutoRcpStatus = Error THEN

				eAutoRcpAct		:= AutoRcpActIdle;
				usiStep			:= 1;

			END_IF

		1:
			eAutoRcpAct	:= AutoRcpActReadRetain;

			IF (p_eAutoRcpStatus = Done) AND (p_eAutoRcpStat = AutoRcpActReadRetain) THEN

				eAutoRcpAct		:= AutoRcpActIdle;
				usiStep			:= 0;
				eStartupStep1	:= StartupStepUsrMgmt;

			ELSIF p_eAutoRcpStatus = Error THEN

				eAutoRcpAct		:= AutoRcpActIdle;
				usiStep			:= 0;
				eStartupStep1	:= StartupStepUsrMgmt;

			END_IF

	END_CASE

END_ACTION
```

#### Act_Main_Recipe.st
```iecst
(** 2019-05-04 **)
ACTION Act_Main_Recipe:

	CASE usiStep OF
		0:
			eProdRcpAct	:= ProdRcpActCreateDir;

			IF (p_eProdRcpStatus = Done) AND (p_eProdRcpStat = ProdRcpActCreateDir) THEN

				eProdRcpAct		:= ProdRcpActIdle;
				usiStep			:= 1;

			ELSIF p_eProdRcpStatus = Error THEN

				eProdRcpAct		:= ProdRcpActIdle;
				usiStep			:= 10;

			END_IF

		1:
			eProdRcpAct	:= ProdRcpActGetList;

			IF (p_eProdRcpStatus = Done) AND (p_eProdRcpStat = ProdRcpActGetList) THEN

				eProdRcpAct		:= ProdRcpActIdle;
				usiStep			:= 2;

			ELSIF p_eProdRcpStatus = Error THEN

				eProdRcpAct		:= ProdRcpActIdle;
				usiStep			:= 10;

			END_IF

		2:
			eProdRcpAct	:= ProdRcpActReadCurrRcp;

			IF (p_eProdRcpStatus = Done) AND (p_eProdRcpStat = ProdRcpActReadCurrRcp) THEN

				eProdRcpAct		:= ProdRcpActIdle;
				usiStep			:= 10;

			ELSIF p_eProdRcpStatus = Error THEN

				eProdRcpAct		:= ProdRcpActIdle;
				usiStep			:= 10;

			END_IF

		10:
			eMpProdRcpAct	:= MpProdRcpActCreateDir;

			IF (p_eMpProdRcpStatus = Done) AND (p_eMpProdRcpStat = MpProdRcpActCreateDir) THEN

				eMpProdRcpAct	:= MpProdRcpActIdle;
				usiStep			:= 20;

			ELSIF p_eProdRcpStatus = Error THEN

				eMpProdRcpAct	:= MpProdRcpActIdle;
				usiStep			:= 20;

			END_IF

		20:
			eMagRcpAct	:= MagRcpActCreateDir;

			IF (p_eMagRcpStatus = Done) AND (p_eMagRcpStat = MagRcpActCreateDir) THEN

				eMagRcpAct		:= MagRcpActIdle;
				usiStep			:= 21;

			ELSIF p_eMagRcpStatus = Error THEN

				eMagRcpAct		:= MagRcpActIdle;
				usiStep			:= 30;

			END_IF

		21:
			eMagRcpAct	:= MagRcpActGetList;

			IF (p_eMagRcpStatus = Done) AND (p_eMagRcpStat = MagRcpActGetList) THEN

				eMagRcpAct		:= MagRcpActIdle;
				usiStep			:= 22;

			ELSIF p_eMagRcpStatus = Error THEN

				eMagRcpAct		:= MagRcpActIdle;
				usiStep			:= 30;

			END_IF

		22:
			eMagRcpAct	:= MagRcpActReadCurrRcp;

			IF (p_eMagRcpStatus = Done) AND (p_eMagRcpStat = MagRcpActReadCurrRcp) THEN

				eMagRcpAct		:= MagRcpActIdle;
				usiStep			:= 30;

			ELSIF p_eMagRcpStatus = Error THEN

				eMagRcpAct		:= MagRcpActIdle;
				usiStep			:= 30;

			END_IF

		30:
			eMagRcpAct1	:= MagRcpActCreateDir;

			IF (p_eMagRcpStatus1 = Done) AND (p_eMagRcpStat1 = MagRcpActCreateDir) THEN

				eMagRcpAct1		:= MagRcpActIdle;
				usiStep			:= 31;

			ELSIF p_eMagRcpStatus1 = Error THEN

				eMagRcpAct1		:= MagRcpActIdle;
				usiStep			:= 0;
				eStartupStep1	:= StartupStepAutoRcp;

			END_IF

		31:
			eMagRcpAct1	:= MagRcpActGetList;

			IF (p_eMagRcpStatus1 = Done) AND (p_eMagRcpStat1 = MagRcpActGetList) THEN

				eMagRcpAct1		:= MagRcpActIdle;
				usiStep			:= 32;

			ELSIF p_eMagRcpStatus1 = Error THEN

				eMagRcpAct1		:= MagRcpActIdle;
				usiStep			:= 0;
				eStartupStep1	:= StartupStepAutoRcp;

			END_IF

		32:
			eMagRcpAct1	:= MagRcpActReadCurrRcp;

			IF (p_eMagRcpStatus1 = Done) AND (p_eMagRcpStat1 = MagRcpActReadCurrRcp) THEN

				eMagRcpAct1		:= MagRcpActIdle;
				usiStep			:= 0;
				eStartupStep1	:= StartupStepAutoRcp;

			ELSIF p_eMagRcpStatus1 = Error THEN

				eMagRcpAct1		:= MagRcpActIdle;
				usiStep			:= 0;
				eStartupStep1	:= StartupStepAutoRcp;

			END_IF

	END_CASE

END_ACTION
```
